METHOD getNewBBSTree :CNM_ReturnTypes.SingleExecutionResult
VAR_INPUT
	(*optional custom comparator*)
	comparator : CNM_AbstractObject.IComparator := 0;
END_VAR
VAR_OUTPUT
	(* the created tree *)
	tree :CNM_CollectionInterfaces.IBalancedBinarySearchTree;
END_VAR 
VAR
	newBalancedBinarySearchTree 	:POINTER TO BalancedBinarySearchTree;
END_VAR
VAR CONSTANT
	OBJECT_NOT_REFERENCED 			:__XWORD		:= 0;
END_VAR
getNewBBSTree := CNM_ReturnTypes.SingleExecutionResult.ERROR;
IF THIS^.isObjectValid(comparator) THEN
	newBalancedBinarySearchTree := __NEW(
	BalancedBinarySearchTree(nodeComparator := comparator)
	);
ELSE
	newBalancedBinarySearchTree := __NEW(
	BalancedBinarySearchTree(nodeComparator := OBJECT_NOT_REFERENCED)
	);
END_IF

IF (newBalancedBinarySearchTree <> 0) THEN
	tree := newBalancedBinarySearchTree^;
	getNewBBSTree := CNM_ReturnTypes.SingleExecutionResult.SUCCESS;
END_IF
END_METHOD

(*

## Short summary

function to create a new balanced binary searchtree node

.. <legal notes>

legal notes
=================
| SPDX-FileCopyrightText: © 2022 ekvip automation GmbH <info@ekvip.de>
| SPDX-License-Identifier: Apache-2.0
| For details check: Apache-2.0_

.. _Apache-2.0: https://www.apache.org/licenses/LICENSE-2.0

.. </legal notes>


**Return:** ``SingleExecutionResult.SUCCESS``: allocation succesful, output node contains new tree node instance
    ``SingleExecutionResult.ERROR``: error during allocation, output node is NULL

*)

METHOD getNewBBSTreeNode :CNM_ReturnTypes.SingleExecutionResult 
VAR_INPUT
	(* the object that should be wrapped *)
	object :CNM_AbstractObject.IObject;
END_VAR
VAR_OUTPUT
	(* the created tree node container element *)
	node :CNM_CollectionInterfaces.IBalancedBinarySearchTreeNode;
END_VAR
VAR 
	newTreeNode 		:POINTER TO BalancedBinarySearchTreeNode;
END_VAR
VAR CONSTANT
	IS_NOT_REFERENCED 	:__XWORD := 0;
END_VAR
getNewBBSTreeNode := CNM_ReturnTypes.SingleExecutionResult.ERROR;
newTreeNode := __NEW(
	BalancedBinarySearchTreeNode(
		value := object,
		left := IS_NOT_REFERENCED,
		right := IS_NOT_REFERENCED
	)
);
IF (newTreeNode <> 0) THEN
	newTreeNode^.leftChild := IS_NOT_REFERENCED;
	newTreeNode^.rightChild := IS_NOT_REFERENCED;
	node := newTreeNode^;
	getNewBBSTreeNode := CNM_ReturnTypes.SingleExecutionResult.SUCCESS;
END_IF
END_METHOD

(*

## Short summary

Method to create new Instance of DoublyLinkedElements and automatically link with other ellements.
This will affect/change the next and previouse elements !

.. <legal notes>

legal notes
=================
| SPDX-FileCopyrightText: © 2022 ekvip automation GmbH <info@ekvip.de>
| SPDX-License-Identifier: Apache-2.0
| For details check: Apache-2.0_

.. _Apache-2.0: https://www.apache.org/licenses/LICENSE-2.0

.. </legal notes>


**Return:** ``SingleExecutionResult.SUCCESS``: allocation succesful, output element contains new list element instance
    ``SingleExecutionResult.ERROR``: error during allocation, output element is NULL

*)

METHOD getNewDoublyLinkedElement :CNM_ReturnTypes.SingleExecutionResult
VAR_INPUT
	(*the dataobject to be contained inside the element*)
	object					:CNM_AbstractObject.IObject;
	(*the previous element to link to*)
	previousElement			:CNM_CollectionInterfaces.IDoublyLinkedElement;
	(*the next element to link to*)
	nextElement				:CNM_CollectionInterfaces.IDoublyLinkedElement;	
	(*a flag if the link to next and previous should be created*)
	linkElements			:BOOL := TRUE;
END_VAR
VAR_OUTPUT
	(* the created array linked list container element *)
	element :CNM_CollectionInterfaces.IDoublyLinkedElement;
END_VAR
VAR
	newElement		:POINTER TO DoublyLinkedElement;
END_VAR
getNewDoublyLinkedElement := CNM_ReturnTypes.SingleExecutionResult.ERROR;
newElement := __NEW(
	DoublyLinkedElement(
		content		:= object,
		previous	:= previousElement,
		next		:= nextElement
	)
);

IF (newElement <> 0) THEN
	IF (linkElements) THEN
		IF (THIS^.isObjectValid(previousElement)) THEN
			previousElement.next := newElement^;
		END_IF
		IF (THIS^.isObjectValid(nextElement)) THEN
			nextElement.previous := newElement^;
		END_IF	
	END_IF
	element := newElement^;
	getNewDoublyLinkedElement := CNM_ReturnTypes.SingleExecutionResult.SUCCESS;
END_IF
END_METHOD

(*

## Short summary

A method to generate a new LinkedList.

.. <legal notes>

legal notes
=================
| SPDX-FileCopyrightText: © 2022 ekvip automation GmbH <info@ekvip.de>
| SPDX-License-Identifier: Apache-2.0
| For details check: Apache-2.0_

.. _Apache-2.0: https://www.apache.org/licenses/LICENSE-2.0

.. </legal notes>



*)

METHOD getNewLinkedList :CNM_ReturnTypes.SingleExecutionResult
VAR_OUTPUT
	(* the created linked list *)
	list :CNM_CollectionInterfaces.ILinkedList;
END_VAR
VAR
	newList	:POINTER TO LinkedList;
END_VAR
getNewLinkedList := CNM_ReturnTypes.SingleExecutionResult.ERROR;
newList := __NEW(
	LinkedList()
);
IF (newList <> 0) THEN
	list := newList^;
	getNewLinkedList := CNM_ReturnTypes.SingleExecutionResult.SUCCESS;
END_IF
END_METHOD

(*

## Short summary

This method will create a new MergeSorter for linked lists.

.. <legal notes>

legal notes
=================
| SPDX-FileCopyrightText: © 2025 ekvip automation GmbH <info@ekvip.de>
| SPDX-License-Identifier: Apache-2.0
| For details check: Apache-2.0_

.. _Apache-2.0: https://www.apache.org/licenses/LICENSE-2.0

.. </legal notes>



*)
METHOD getNewLinkedListMergeSorter : CNM_CollectionInterfaces.CNM_ReturnTypes.SingleExecutionResult
VAR_OUTPUT
	(* the created linked list merge sorter *)
	sorter	: CNM_CollectionInterfaces.ILinkedListSorter;
END_VAR
VAR
	newMergeSorter :POINTER TO LinkedListMergeSorter; 
END_VAR
getNewLinkedListMergeSorter := CNM_ReturnTypes.SingleExecutionResult.ERROR;
newMergeSorter := __NEW(LinkedListMergeSorter());

IF (newMergeSorter <> 0) THEN
	sorter := newMergeSorter^;
	getNewLinkedListMergeSorter := CNM_ReturnTypes.SingleExecutionResult.SUCCESS;
END_IF
END_METHOD

END_FUNCTION_BLOCK

// ---- Lists/ArrayList/ArrayListSorter/ArrayListMergeSorter.TcPOU
(*

## Short summary

This FB sorts the list using a mergesort, which has O(n*log(n)) runtime. 
For random data it is a bit faster than Timsort, else Timsort should be used. Needs to allocate extra memory while sorting, same size as currentContainerSize.

**Caution:**
	Due to the characteristics of a merge, a merge must be performed atomically.
	As a merge of two lists l1 and l2 can take up to l1.size compares.
	That implies that at the last cycle of the merge, an atomic operation that requires up to list.size/2 compares must be performed.
	Therefore the maxCycleCompares may be exceeded and set the maxCycleCompares to a value smaller than list.size/2 may not have the desired effect.
	
.. <legal notes>

legal notes
=================
| SPDX-FileCopyrightText: © 2022 ekvip automation GmbH <info@ekvip.de>
| SPDX-License-Identifier: Apache-2.0
| For details check: Apache-2.0_

.. _Apache-2.0: https://www.apache.org/licenses/LICENSE-2.0

.. </legal notes>



*)

{attribute 'enable_dynamic_creation'}
FUNCTION_BLOCK FINAL ArrayListMergeSorter EXTENDS AbstractMergeBasedSorter
VAR
	sortBuffer :POINTER TO CNM_AbstractObject.IObject;
END_VAR


(*

## Short summary

This abstract property returns the class name of the concrete object, 
which is useful to check the class name for ``__DELETE``.

.. <legal notes>

legal notes
=================
| SPDX-FileCopyrightText: © 2022 ekvip automation GmbH <info@ekvip.de>
| SPDX-License-Identifier: Apache-2.0
| For details check: Apache-2.0_

.. _Apache-2.0: https://www.apache.org/licenses/LICENSE-2.0

.. </legal notes>

*)
PROPERTY className	:CNM_AbstractObject.ClassName
GET
className := 'CNM_Collections.ArrayListMergeSorter';
END_GET
END_PROPERTY


(*

## Short summary

This method is used to create a new instance
of the object which has the same internal state as the object.
If the object is a container class, the references to the content objects
are not cloned for this there is the method ``ICloneable.deepClone``.

If an object does not support cloning the return value is
``CNM_ReturnTypes.CloneResult.CLONE_IS_NOT_SUPPORTED``.

If there is not enough memory or the cloning fails because the
attribute enable dynamic creation was forgotten the return value is 
``CNM_ReturnTypes.CloneResult.FAILED``.

Only if the return value is ``CNM_ReturnTypes.CloneResult.SUCCESS``
the output ``clonedObject`` points to the new object
otherwise ``clonedObject`` is NULL.  

.. <legal notes>

legal notes
=================
| SPDX-FileCopyrightText: © 2022 ekvip automation GmbH <info@ekvip.de>
| SPDX-License-Identifier: Apache-2.0
| For details check: Apache-2.0_

.. _Apache-2.0: https://www.apache.org/licenses/LICENSE-2.0

.. </legal notes>


**Return:**	``CNM_ReturnTypes.CloneResult.SUCCESS``: new object clone was created,
	``CNM_ReturnTypes.CloneResult.FAILED``: object clone failed
	``CNM_ReturnTypes.CloneResult.CLONE_IS_NOT_SUPPORTED``: object does not support cloning

*)
METHOD clone	:CNM_AbstractObject.CNM_ReturnTypes.CloneResult
VAR_OUTPUT
	(* new object instance or NULL if somthing went wrong *)
	clonedObject	:CNM_AbstractObject.IObject;
END_VAR
VAR
	newSorter :POINTER TO ArrayListMergeSorter;
	sorter :CNM_CollectionInterfaces.IArrayListSorter;
END_VAR
newSorter := __NEW(
	ArrayListMergeSorter()
);

IF (newSorter = 0) THEN
	clone := CNM_ReturnTypes.CloneResult.FAILED;
ELSE
	clone := CNM_ReturnTypes.CloneResult.SUCCESS;
	THIS^.prepareClonedSorter(newSorter^);
	clonedObject := newSorter^;
END_IF
END_METHOD

(*

## Short summary

Mark the object as deleted, as it staiys in the memory.

.. <legal notes>

legal notes
=================
| SPDX-FileCopyrightText: © 2022 ekvip automation GmbH <info@ekvip.de>
| SPDX-License-Identifier: Apache-2.0
| For details check: Apache-2.0_

.. _Apache-2.0: https://www.apache.org/licenses/LICENSE-2.0

.. </legal notes>

*)
METHOD FB_Exit : BOOL
VAR_INPUT
	(* TRUE: the exit method is called in order to leave the instance which will be copied afterwards (online change).*)
	bInCopyCode	: BOOL;
END_VAR
IF THIS^.sortBuffer <> 0  THEN
	__DELETE(THIS^.sortBuffer);	
END_IF
END_METHOD

(*

## Short summary

This method sorts the data structure instantly within one call. 
It uses the passed Comparator to sort the structure or the compareTo of the contained Objects if no comparator is passed.

.. <legal notes>

legal notes
=================
| SPDX-FileCopyrightText: © 2022 ekvip automation GmbH <info@ekvip.de>
| SPDX-License-Identifier: Apache-2.0
| For details check: Apache-2.0_

.. _Apache-2.0: https://www.apache.org/licenses/LICENSE-2.0

.. </legal notes>


**Return:**``ERROR``: Sort was not able to finish 
	``SUCCESS``: Sorting was finished succesfully

*)
METHOD instantSort : CNM_CollectionInterfaces.CNM_ReturnTypes.SingleExecutionResult
VAR_INPUT
	(*The size of the list to be sorted*)
	size	: UDINT;
	(*the container, that contains the list elements*)
	container	: POINTER TO CNM_CollectionInterfaces.CNM_AbstractObject.IObject;
	(*the comparator that should be used for the sort. Must not be changed while sort is in process*)
	comparator	: CNM_CollectionInterfaces.CNM_AbstractObject.IComparator := 0;
END_VAR
VAR_IN_OUT
	(*the current version of the list, must change when the data in the list changes *)
	currentListVersion	: __XWORD;
END_VAR
VAR 
	instantSortBuffer :POINTER TO CNM_AbstractObject.IObject;
	currentSortSize 	:UDINT := 1;
	leftBound 			:UDINT;
	middle 				:UDINT;
	rightBound 			:UDINT;
	maximumLeftBound	:UDINT;
	stepSize 			:UDINT;
END_VAR
VAR CONSTANT
	NULL :__XWORD := 0;
END_VAR
instantSortBuffer := __NEW(__XWORD, size);
THIS^.setComparator(comparator);
WHILE (currentSortSize <= size-1) DO
	maximumLeftBound := size -2;
	stepSize := 2*currentSortSize;
	FOR leftBound := 0 TO maximumLeftBound BY (stepSize) DO
		
		IF leftBound+currentSortSize-1 < size-1 THEN
			middle := leftBound + currentSortSize-1;
		ELSE
			middle := size-1;
		END_IF
		IF leftBound + stepSize - 1 < size THEN
			rightBound := leftBound + stepSize -1;
		ELSE
			rightBound := size-1;
		END_IF
		
		instantSort := merge(
			firstContainer := ADR(container[leftBound]),
			secondContainer := ADR(container[middle + 1]),
			buffer := instantSortBuffer,
			firstContainerSize := middle - leftBound + 1,
			secondContainerSize := rightBound - middle 
		);
		IF instantSort <> CNM_ReturnTypes.SingleExecutionResult.SUCCESS THEN
			__DELETE(instantSortBuffer);
			RETURN;
		END_IF
		
		Tc2_System.MEMMOVE(
			destAddr := ADR(container[leftBound]),
			srcAddr := THIS^.sortBuffer,
			n := rightBound - leftBound + 1
		);
	END_FOR
END_WHILE

currentListVersion := currentListVersion + 1;
instantSort := CNM_ReturnTypes.SingleExecutionResult.SUCCESS;
END_METHOD

(*

## Short summary

This method sorts the data structure. 
It uses the passed Comperator to sort the structure.
This can take many cycles and should be called until the CNM_ReturnTypes.ExecutionState is no longer ``BUSY``.

.. <legal notes>

legal notes
=================
| SPDX-FileCopyrightText: © 2022 ekvip automation GmbH <info@ekvip.de>
| SPDX-License-Identifier: Apache-2.0
| For details check: Apache-2.0_

.. _Apache-2.0: https://www.apache.org/licenses/LICENSE-2.0

.. </legal notes>


**Return:** ``ABORTED``: While sort was pending,execute had a falling edge,
	``BUSY``: Sort is in progress
	``ERROR``: Sort was not able to finish (p.e. List changed) call sort(false) to reset
	``IDLE``: Currently no sort in progress
	``SUCCESS``: Sorting was finished 

*)
METHOD sort	:CNM_ReturnTypes.SingleExecutionState
VAR_INPUT
	(*control bit to start or abort the sorting, needs to be active until the ExecutionState is SUCCESS*)
	execute		:BOOL;
	(*The size of the list to be sorted*)
	size 		:UDINT;
	(*the container, that contains the list elements*)
	container	:POINTER TO CNM_AbstractObject.IObject;
	(*the comparator that should be used for the sort. Must not be changed while sort is in process*)
	comparator	:CNM_AbstractObject.IComparator		:= 0;
END_VAR
VAR_IN_OUT
	(*the current version of the list, must change when the data in the list changes *)
	currentListVersion :__XWORD;
END_VAR
VAR_INST
	cycleManager :CNM_CycleManager.SimpleCycleManager;
	lastExecute			:BOOL		:= FALSE;
	executing 			:BOOL		:= FALSE;
	state 				:CNM_ReturnTypes.SingleExecutionState	:= CNM_ReturnTypes.SingleExecutionState.IDLE; 
	currentSortSize 	:UDINT;
	startAt 			:UDINT 	:= 0;
	(* list version index, used to detect list changes during sorting *)
	lastListChangeIndex :__XWORD;
END_VAR
VAR 
	leftBound 			:UDINT;
	middle 				:UDINT;
	rightBound 			:UDINT;
	operationsThisCycle	:UDINT :=0;
	leave 				:BOOL := FALSE;
	mergeState 			:CNM_ReturnTypes.SingleExecutionResult;
	maximumLeftBound	:UDINT;
	stepSize 			:UDINT;
END_VAR
VAR CONSTANT
	INIT :DINT := CNM_ReturnTypes.DefaultSteps.STEP.INIT;
	SORT_LIST :DINT := INIT + 1;
	CLEAN_UP :DINT := SORT_LIST + 1;
	ERROR :DINT := CNM_ReturnTypes.DefaultSteps.STEP.ERROR;
	REGISTER_SIZE :UDINT := SIZEOF(__XWORD);
END_VAR
cycleManager(execute := execute);
IF cycleManager.step.current > INIT THEN
	cycleManager.assert.bitNumber.x.valueIsEqualTo(
		currentValue := currentListVersion, 
		expectedValue := lastListChangeIndex, 
		message := 'list has changed during pending sorting'
	);
END_IF


CASE cycleManager.step.current OF
INIT:
	cycleManager.configuration.sequence.requireSuccessStep := FALSE;
	THIS^.setComparator(comparator);
	lastListChangeIndex := currentListVersion;
	startAt := 0;
	IF size > 1 THEN
		currentSortSize := 1;
		__DELETE(THIS^.sortBuffer);
		THIS^.sortBuffer := __NEW(__XWORD, size);
		THIS^.maxOperationsPerCycle := size;
		cycleManager.proceed();
	ELSE
		cycleManager.proceedWith(step := CNM_ReturnTypes.DefaultSteps.STEP.SUCCESS);
	END_IF
	
SORT_LIST:
	IF (lastListChangeIndex <> currentListVersion) THEN
		cycleManager.proceedWith(ERROR);
		sort := CNM_ReturnTypes.SingleExecutionState.ERROR;
		RETURN;
	END_IF
	IF currentSortSize <= size-1 THEN
		WHILE (operationsThisCycle < THIS^.maxCycleCompares) DO
			maximumLeftBound := size -2;
			stepSize := 2*currentSortSize;
			FOR leftBound := startAt TO maximumLeftBound BY (stepSize) DO
				IF (operationsThisCycle > THIS^.maxCycleCompares) THEN
					leave := TRUE;
					EXIT;
				END_IF
				
				IF leftBound+currentSortSize-1 < size-1 THEN
					middle := leftBound + currentSortSize-1;
				ELSE
					middle := size-1;
				END_IF
				IF leftBound + stepSize - 1 < size THEN
					rightBound := leftBound + stepSize -1;
				ELSE
					rightBound := size-1;
				END_IF
				
				mergeState := merge(
					firstContainer := ADR(container[leftBound]),
					secondContainer := ADR(container[middle + 1]),
					buffer := THIS^.sortBuffer,
					firstContainerSize := middle - leftBound + 1,
					secondContainerSize := rightBound - middle 
				);
				IF mergeState <> CNM_ReturnTypes.SingleExecutionResult.SUCCESS THEN
					cycleManager.proceedWith(CNM_ReturnTypes.DefaultSteps.STEP.ERROR);
					sort := CNM_ReturnTypes.SingleExecutionState.ERROR;
					RETURN;
				END_IF
				Tc2_System.MEMMOVE(
					destAddr := ADR(container[leftBound]),
					srcAddr := THIS^.sortBuffer,
					n := (rightBound - leftBound + 1) * REGISTER_SIZE
				);
				operationsThisCycle := operationsThisCycle + stepSize - 1;
				
			END_FOR
			
			IF leave THEN
				startAt := leftBound;
				EXIT;
			ELSE
				startAt := 0;
				currentSortSize := stepSize;
				IF currentSortSize > size-1 THEN
					EXIT;
				END_IF
			END_IF
		END_WHILE
	END_IF

	//check if sort done within same cycle
	IF currentSortSize > size-1 THEN 
		cycleManager.proceedWith(CNM_ReturnTypes.DefaultSteps.STEP.SUCCESS);
		IF THIS^.sortBuffer <> 0  THEN
			__DELETE(sortBuffer);	
		END_IF
	END_IF
	
	lastListChangeIndex := currentListVersion := currentListVersion + 1;
	
CLEAN_UP,
CNM_ReturnTypes.DefaultSteps.STEP.ERROR,
CNM_ReturnTypes.DefaultSteps.STEP.ABORT,
CNM_ReturnTypes.DefaultSteps.STEP.SUCCESS:
	IF THIS^.sortBuffer <> 0  THEN
		__DELETE(sortBuffer);	
	END_IF
	
END_CASE
sort := cycleManager.state;
END_METHOD

END_FUNCTION_BLOCK

// ---- Lists/ArrayList/ArrayListSorter/AbstractMergeBasedSorter.TcPOU
(*

## Short summary

Abstract Sorter for merge based sort methods. 
Provides a default implementation for an indexed merge function and a method to efficient copy elements.

**Caution:**
	Due to the characteristics of a merge, a merge must be performed atomically.
	As a merge of two lists l1 and l2 can take up to l1.size+l2.size-1 compares.
	That implies that at the last cycle of the merge, an atomic operation that requires up to list.size-1 compares must be performed.
	Therefore the maxCycleCompares may be exceeded and set the maxCycleCompares to a value smaller than list.size-1 may not have the desired effect.
 
.. <legal notes>

legal notes
=================
| SPDX-FileCopyrightText: © 2022 ekvip automation GmbH <info@ekvip.de>
| SPDX-License-Identifier: Apache-2.0
| For details check: Apache-2.0_

.. _Apache-2.0: https://www.apache.org/licenses/LICENSE-2.0

.. </legal notes>



*)

FUNCTION_BLOCK INTERNAL ABSTRACT AbstractMergeBasedSorter EXTENDS AbstractArrayListSorter

(*

## Short summary

Function that sorts specified parts using a merge mechanism.
Writes the result into a given buffer. 
Buffer size must be at least as big as both given containers combined.

.. <legal notes>

legal notes
=================
| SPDX-FileCopyrightText: © 2025 ekvip automation GmbH <info@ekvip.de>
| SPDX-License-Identifier: Apache-2.0
| For details check: Apache-2.0_

.. _Apache-2.0: https://www.apache.org/licenses/LICENSE-2.0

.. </legal notes>


**Return:** CNM_ReturnTypes.ExecutionResult: the result of the merge,
	ERROR if any parameter was invalid for merge 
	SUCCESS if list is merged and result in buffer

*)

METHOD PROTECTED FINAL merge : CNM_ReturnTypes.SingleExecutionResult
VAR_INPUT
	firstContainer :POINTER TO CNM_AbstractObject.IObject;
	secondContainer :POINTER TO CNM_AbstractObject.IObject;
	buffer :POINTER TO CNM_AbstractObject.IObject;
	firstContainerSize :UDINT;
	secondContainerSize :UDINT;
END_VAR
VAR
	leftIndex :UDINT;
	rightIndex :UDINT;
	destination :__XWORD;
	source :__XWORD;
	remainingElements :UDINT;
END_VAR
VAR CONSTANT
	REGISTER_SIZE :UDINT := SIZEOF(__XWORD);
END_VAR
merge := CNM_ReturnTypes.SingleExecutionResult.ERROR;
RETURN (
	(buffer = 0)
	OR_ELSE (firstContainer = 0) 
	OR_ELSE (secondContainer = 0)
	OR_ELSE (firstContainer = secondContainer)
);

merge := CNM_ReturnTypes.SingleExecutionResult.SUCCESS;
RETURN (
	((firstContainerSize + secondContainerSize) = 0) 
);

WHILE(
	(rightIndex < secondContainerSize) 
	AND_THEN (leftIndex < firstContainerSize)
)DO
	IF ( 
		THIS^.compareElements(
			firstContainer[leftIndex],secondContainer[rightIndex]
		) <= CNM_ReturnTypes.ComparationResult.EQUAL
	) THEN
		buffer[leftIndex+rightIndex] := firstContainer[leftIndex];
		leftIndex := leftIndex + 1;
	ELSE
		buffer[leftIndex+rightIndex] := secondContainer[rightIndex];
		rightIndex := rightIndex + 1;
	END_IF
END_WHILE

destination := ADR(buffer[leftIndex+rightIndex]);
IF(leftIndex = firstContainerSize)THEN
	source := ADR(secondContainer[rightIndex]);
	remainingElements := secondContainerSize - rightIndex;
ELSE
	source := ADR(firstContainer[leftIndex]);
	remainingElements := firstContainerSize - leftIndex;
END_IF

Tc2_System.MEMMOVE(
	destAddr := destination,
	srcAddr := source,
	n := remainingElements * REGISTER_SIZE
);
END_METHOD

END_FUNCTION_BLOCK

// ---- Lists/Sorter/classes/AbstractArrayListSorter.TcPOU
(*

## Short summary

The abstract implementation of an ArrayListSorter, to provide default implementations for setting comparator, the IObject methods.
Provides the default implementation for sort and inverseSort.

.. <legal notes>

legal notes
=================
| SPDX-FileCopyrightText: © 2022 ekvip automation GmbH <info@ekvip.de>
| SPDX-License-Identifier: Apache-2.0
| For details check: Apache-2.0_

.. _Apache-2.0: https://www.apache.org/licenses/LICENSE-2.0

.. </legal notes>



*)

FUNCTION_BLOCK INTERNAL ABSTRACT AbstractArrayListSorter EXTENDS AbstractListSorter IMPLEMENTS CNM_CollectionInterfaces.IArrayListSorter

(*

## Short summary

This method sorts the data structure instantly in descending order within one call. 
It uses the passed Comparator to sort the structure or the compareTo of the contained Objects if no comparator is passed.

.. <legal notes>

legal notes
=================
| SPDX-FileCopyrightText: © 2022 ekvip automation GmbH <info@ekvip.de>
| SPDX-License-Identifier: Apache-2.0
| For details check: Apache-2.0_

.. _Apache-2.0: https://www.apache.org/licenses/LICENSE-2.0

.. </legal notes>


**Return:**``ERROR``: Sort was not able to finish 
	``SUCCESS``: Sorting was finished succesfully

*)
METHOD instantInverseSort : CNM_CollectionInterfaces.CNM_ReturnTypes.SingleExecutionResult
VAR_INPUT
	(*The size of the list to be sorted*)
	size	: UDINT;
	(*the container, that contains the list elements*)
	container	: POINTER TO CNM_CollectionInterfaces.CNM_AbstractObject.IObject;
	(*the comparator that should be used for the sort. Must not be changed while sort is in process*)
	comparator	: CNM_CollectionInterfaces.CNM_AbstractObject.IComparator := 0;
END_VAR
VAR_IN_OUT
	(*the current version of the list, must change when the data in the list changes *)
	currentListVersion	: __XWORD;
END_VAR
THIS^.reverseComparator.attachComparator(comparator);
THIS^.instantSort(size := size, comparator := THIS^.reverseComparator, container := container, currentListVersion := currentListVersion);
END_METHOD

(*

## Short summary

This method sorts the data structure instantly within one call. 
It uses the passed Comparator to sort the structure or the compareTo of the contained Objects if no comparator is passed.

.. <legal notes>

legal notes
=================
| SPDX-FileCopyrightText: © 2022 ekvip automation GmbH <info@ekvip.de>
| SPDX-License-Identifier: Apache-2.0
| For details check: Apache-2.0_

.. _Apache-2.0: https://www.apache.org/licenses/LICENSE-2.0

.. </legal notes>


**Return:**``ERROR``: Sort was not able to finish 
	``SUCCESS``: Sorting was finished succesfully

*)
METHOD ABSTRACT instantSort : CNM_CollectionInterfaces.CNM_ReturnTypes.SingleExecutionResult
VAR_INPUT
	(*The size of the list to be sorted*)
	size	: UDINT;
	(*the container, that contains the list elements*)
	container	: POINTER TO CNM_CollectionInterfaces.CNM_AbstractObject.IObject;
	(*the comparator that should be used for the sort. Must not be changed while sort is in process*)
	comparator	: CNM_CollectionInterfaces.CNM_AbstractObject.IComparator := 0;
END_VAR
VAR_IN_OUT
	(*the current version of the list, must change when the data in the list changes *)
	currentListVersion	: __XWORD;
END_VAR
END_METHOD


(*

## Short summary

This method sorts the Sortable in the inverted order, so from great to low
.. <legal notes>

legal notes
=================
| SPDX-FileCopyrightText: © 2025 ekvip automation GmbH <info@ekvip.de>
| SPDX-License-Identifier: Apache-2.0
| For details check: Apache-2.0_

.. _Apache-2.0: https://www.apache.org/licenses/LICENSE-2.0

.. </legal notes>


**Return:** ``ABORTED``: While inverse was pending,execute had a falling edge,
	``BUSY``: Inverse is in progress
	``ERROR``: Inverse was not able to finish (p.e. List changed) call inverse(false) to reset
	``IDLE``: Currently invert is not in progress
	``SUCCESS``: Inversing was finished 
*)
METHOD inverseSort : CNM_ReturnTypes.SingleExecutionState
VAR_INPUT
	(*control bit to start or abort the inverting, needs to be active until the ExecutionState is noz longer busy*)
	execute	: BOOL;
	(*The size of the list to be sorted*)
	size :UDINT;
	(*the container, that contains the list elements*)
	container	: POINTER TO CNM_AbstractObject.IObject;
END_VAR
VAR_INPUT
	(*the comparator that should be used for the sort. Must not be changed while sort is in process*)
	comparator :CNM_AbstractObject.IComparator := 0;
END_VAR
VAR_IN_OUT
	(*the current version of the list, must change when the data in the list changes *)
	currentListVersion :__XWORD;
END_VAR
THIS^.reverseComparator.attachComparator(comparator);
THIS^.sort(execute := execute, size := size, comparator := THIS^.reverseComparator, container := container, currentListVersion := currentListVersion);
END_METHOD

(*

## Short summary

This method sorts the data structure. 
This can take many cycles and should be called until the CNM_ReturnTypes.ExecutionState is no longer ``BUSY``.

.. <legal notes>

legal notes
=================
| SPDX-FileCopyrightText: © 2025 ekvip automation GmbH <info@ekvip.de>
| SPDX-License-Identifier: Apache-2.0
| For details check: Apache-2.0_

.. _Apache-2.0: https://www.apache.org/licenses/LICENSE-2.0

.. </legal notes>


**Return:** ``ABORTED``: While sort was pending,execute had a falling edge,
	``BUSY``: Sort is in progress
	``ERROR``: Sort was not able to finish (p.e. List changed) call sort(false) to reset
	``IDLE``: Currently no sort in progress
	``SUCCESS``: Sorting was finished 

*)
METHOD ABSTRACT sort :CNM_ReturnTypes.SingleExecutionState
VAR_INPUT
	(*control bit to start or abort the sorting, needs to be active until the ExecutionState is SUCCESS*)
	execute		:BOOL;
	(*The size of the list to be sorted*)
	size 		:UDINT;
	(*the container, that contains the list elements*)
	container	:POINTER TO CNM_AbstractObject.IObject;
	(*the comparator that should be used for the sort. Must not be changed while sort is in process*)
	comparator :CNM_AbstractObject.IComparator := 0;
END_VAR
VAR_IN_OUT
	(*the current version of the list, must change when the data in the list changes *)
	currentListVersion :__XWORD;
END_VAR
END_METHOD

END_FUNCTION_BLOCK

// ---- Lists/Sorter/classes/AbstractListSorter.TcPOU
(*

## Short summary

Abstract base class for list sorters. Provides functionality to set the execution limits, size and list changes.

.. <legal notes>

legal notes
=================
| SPDX-FileCopyrightText: © 2023 ekvip automation GmbH <info@ekvip.de>
| SPDX-License-Identifier: Apache-2.0
| For details check: Apache-2.0_

.. _Apache-2.0: https://www.apache.org/licenses/LICENSE-2.0

.. </legal notes>



*)

FUNCTION_BLOCK INTERNAL ABSTRACT AbstractListSorter EXTENDS AbstractDisposableContainer IMPLEMENTS CNM_CollectionInterfaces.IListSorter
VAR
	(*The comparator used to sort, set by the List when setting sorter*)
	elementComparator		:CNM_AbstractObject.IComparator;
	(*The maximum of comparisons that the sorter allows, may be overwruled by the bounds*)
	maxOperationsPerCycle 	:UDINT;
	(*The maximum of compares done per cycle to prevent very long lists to take up to much time*)
	upperCompareBound 		:UDINT	:= GeneralParameters.DEFAULT_OPERATIONS_PER_CYCLE;
	(* Comparator used for inverse Sort *)
	reverseComparator :InvertComparator;
	(* the current change index of the list *)
	listChangeIndex :REFERENCE TO __XWORD;
END_VAR


(*

## Short summary

This abstract property returns the class name of the concrete object, 
which is useful to check the class name for ``__DELETE``.

.. <legal notes>

legal notes
=================
| SPDX-FileCopyrightText: © 2022 ekvip automation GmbH <info@ekvip.de>
| SPDX-License-Identifier: Apache-2.0
| For details check: Apache-2.0_

.. _Apache-2.0: https://www.apache.org/licenses/LICENSE-2.0

.. </legal notes>

*)
PROPERTY ABSTRACT className	:CNM_AbstractObject.ClassName
GET
END_GET
END_PROPERTY

(*

## Short summary

This method is called in the destruct method and is intended to zero all references and interfaces that should not be destructed. 
To delete the collection with all its contents, use deepDestruct() instead of destruct().

.. <legal notes>

legal notes
=================
| SPDX-FileCopyrightText: © 2025 ekvip automation GmbH <info@ekvip.de>
| SPDX-License-Identifier: Apache-2.0
| For details check: Apache-2.0_

.. _Apache-2.0: https://www.apache.org/licenses/LICENSE-2.0

.. </legal notes>

*)
METHOD PROTECTED clearContents
THIS^.elementComparator := 0;
END_METHOD


(*

## Short summary

This method is used to create a new instance
of the object which has the same internal state as the object.
If the object is a container class, the references to the content objects
are not cloned for this there is the method `ICloneable.deepClone`.

If an object does not support cloning the return value is
``CNM_ReturnTypes.CloneResult.CLONE_IS_NOT_SUPPORTED``.

If there is not enough memory or the cloning fails because the
attribute enable dynamic creation was forgotten the return value is 
``CNM_ReturnTypes.CloneResult.FAILED``.

Only if the return value is ``CNM_ReturnTypes.CloneResult.SUCCESS``
the output ``clonedObject`` points to the new object
otherwise ``clonedObject`` is NULL.  

.. <legal notes>

legal notes
=================
| SPDX-FileCopyrightText: © 2022 ekvip automation GmbH <info@ekvip.de>
| SPDX-License-Identifier: Apache-2.0
| For details check: Apache-2.0_

.. _Apache-2.0: https://www.apache.org/licenses/LICENSE-2.0

.. </legal notes>


**Return:** ``CNM_ReturnTypes.CloneResult.SUCCESS``: new object clone was created,
    ``CNM_ReturnTypes.CloneResult.FAILED``: object clone failed
    ``CNM_ReturnTypes.CloneResult.CLONE_IS_NOT_SUPPORTED``: object does not support cloning

*)

METHOD ABSTRACT clone	:CNM_AbstractObject.CNM_ReturnTypes.CloneResult
VAR_OUTPUT
	(* new object instance or NULL if somthing went wrong *)
	clonedObject	:CNM_AbstractObject.IObject;
END_VAR
END_METHOD

(*

## Short summary

Compares two objects, if set uses the comparator, else uses the built in comparator of object1.

.. <legal notes>

legal notes
=================
| SPDX-FileCopyrightText: © 2022 ekvip automation GmbH <info@ekvip.de>
| SPDX-License-Identifier: Apache-2.0
| For details check: Apache-2.0_

.. _Apache-2.0: https://www.apache.org/licenses/LICENSE-2.0

.. </legal notes>


**Return:** ``Smaller``: ``Object1`` precendes ``Object2`` in order,
	``Greater``: ``Object1`` succeds ``Object2`` in order,
	``Equal``: ``Object1`` equals ``Object2`` in Order
	
*)

METHOD PROTECTED compareElements	:CNM_ReturnTypes.ComparationResult
VAR_INPUT
	(*first object to compare*)
	object1	:CNM_AbstractObject.IObject;
	(*second object to compare*)
	object2	:CNM_AbstractObject.IObject;
END_VAR
IF THIS^.isObjectValid(THIS^.elementComparator) THEN 
	compareElements := THIS^.elementComparator.compare(object1,object2);   
ELSIF (THIS^.isObjectValid(object1)) THEN
	compareElements := object1.compareTo(object2);
ELSIF (THIS^.isObjectValid(object2)) THEN
	compareElements := CNM_ReturnTypes.ComparationResult.GREATER;
ELSE
	compareElements := CNM_ReturnTypes.ComparationResult.EQUAL;
END_IF
END_METHOD


(*

## Short summary

This method is used to create a new instance
of the object which has the same internal state as the object.
If the object is a container class, the references to the content objects
are cloned too.

If an object does not support cloning the return value is
``CNM_ReturnTypes.CloneResult.CLONE_IS_NOT_SUPPORTED``.

If there is not enough memory or the cloning fails because the
attribute enable dynamic creation was forgotten the return value is 
``CNM_ReturnTypes.CloneResult.FAILED``.
If something goes wrong, then this method must clean up everything
that has been cloned and free the memory again.
**The deepClone either works completely, or not at all**

Only if the return value is ``CNM_ReturnTypes.CloneResult.SUCCESS``
the output ``clonedObject`` points to the new object
otherwise ``clonedObject`` is NULL.  

.. <legal notes>

legal notes
=================
| SPDX-FileCopyrightText: © 2022 ekvip automation GmbH <info@ekvip.de>
| SPDX-License-Identifier: Apache-2.0
| For details check: Apache-2.0_

.. _Apache-2.0: https://www.apache.org/licenses/LICENSE-2.0

.. </legal notes>


**Return:** ``CNM_ReturnTypes.CloneResult.SUCCESS``: new object clone was created,
    ``CNM_ReturnTypes.CloneResult.FAILED``: object clone failed
    ``CNM_ReturnTypes.CloneResult.CLONE_IS_NOT_SUPPORTED``: object does not support deep cloning

*)

METHOD deepClone	:CNM_AbstractObject.CNM_ReturnTypes.CloneResult
VAR_OUTPUT
	(* new object instance or NULL if somthing went wrong *)
	clonedObject	:CNM_AbstractObject.IObject;
END_VAR
deepClone := THIS^.clone(clonedObject => clonedObject);
END_METHOD

(*

## Short summary

Mark the object as deleted, as it staiys in the memory.

.. <legal notes>

legal notes
=================
| SPDX-FileCopyrightText: © 2022 ekvip automation GmbH <info@ekvip.de>
| SPDX-License-Identifier: Apache-2.0
| For details check: Apache-2.0_

.. _Apache-2.0: https://www.apache.org/licenses/LICENSE-2.0

.. </legal notes>

*)
METHOD FB_Exit : BOOL
VAR_INPUT
	(* TRUE: the exit method is called in order to leave the instance which will be copied afterwards (online change).*)
	bInCopyCode	: BOOL;
END_VAR
IF THIS^.isObjectValid(THIS^.elementComparator) THEN
	THIS^.elementComparator.deepDestruct();
END_IF
END_METHOD

(*

## Short summary

This property defines the maximum amount of compares that should be done per Cycle. Is optional as default should be set by class.
Passing zero resets to class specific default.

.. <legal notes>

legal notes
=================
| SPDX-FileCopyrightText: © 2022 ekvip automation GmbH <info@ekvip.de>
| SPDX-License-Identifier: Apache-2.0
| For details check: Apache-2.0_

.. _Apache-2.0: https://www.apache.org/licenses/LICENSE-2.0

.. </legal notes>

*)

PROPERTY maxCycleCompares	:UDINT
GET
maxCycleCompares := THIS^.upperCompareBound;
END_GET
SET
THIS^.upperCompareBound := SEL(
	maxCycleCompares = 0,
	maxCycleCompares,
	GeneralParameters.DEFAULT_OPERATIONS_PER_CYCLE
);
END_SET
END_PROPERTY

(*

## Short summary

Does the basic initialization for a new sorter that was cloned from THIS^

.. <legal notes>

legal notes
=================
| SPDX-FileCopyrightText: © 2022 ekvip automation GmbH <info@ekvip.de>
| SPDX-License-Identifier: Apache-2.0
| For details check: Apache-2.0_

.. _Apache-2.0: https://www.apache.org/licenses/LICENSE-2.0

.. </legal notes>



*)

METHOD PROTECTED prepareClonedSorter
VAR_INPUT
	(*The cloned sorter to init*)
	newSorter :CNM_CollectionInterfaces.IListSorter;
END_VAR
IF (THIS^.isObjectValid(newSorter)) THEN
	newSorter.maxCycleCompares := THIS^.maxCycleCompares;	
END_IF
END_METHOD

(*

## Short summary

This method can replace the default comperator for custom one.
Useful if you par example want to invert the order of the sort.

.. <legal notes>

legal notes
=================
| SPDX-FileCopyrightText: © 2022 ekvip automation GmbH <info@ekvip.de>
| SPDX-License-Identifier: Apache-2.0
| For details check: Apache-2.0_

.. _Apache-2.0: https://www.apache.org/licenses/LICENSE-2.0

.. </legal notes>


**Return:** ``THIS^`` `IListSorter`

*)

METHOD PROTECTED setComparator	:CNM_CollectionInterfaces.IListSorter
VAR_INPUT
	(*the instance of the comperator to be used for sorting*)
	comparator	:CNM_AbstractObject.IComparator;
END_VAR
THIS^.elementComparator := comparator;
setComparator := THIS^;
END_METHOD

END_FUNCTION_BLOCK

// ---- Lists/Sorter/classes/Internal/InvertComparator.TcPOU
(*

## Short summary

Internal comparator, which returns the opposite of the .compareTo method of object1.


.. <legal notes>

legal notes
=================
| SPDX-FileCopyrightText: © 2024 ekvip automation GmbH <info@ekvip.de>
| SPDX-License-Identifier: Apache-2.0
| For details check: Apache-2.0_

.. _Apache-2.0: https://www.apache.org/licenses/LICENSE-2.0

.. </legal notes>



*)

FUNCTION_BLOCK INTERNAL InvertComparator EXTENDS CNM_AbstractObject.Object IMPLEMENTS CNM_AbstractObject.IComparator
VAR
	comparator :CNM_AbstractObject.IComparator;
END_VAR

METHOD attachComparator
VAR_INPUT
	comparator :CNM_AbstractObject.IComparator;
END_VAR
THIS^.comparator := comparator;
END_METHOD


(*

## Short summary

This abstract property returns the class name of the concrete object, 
which is useful to check the class name for ``__DELETE``.

.. <legal notes>

legal notes
=================
| SPDX-FileCopyrightText: © 2022 ekvip automation GmbH <info@ekvip.de>
| SPDX-License-Identifier: Apache-2.0
| For details check: Apache-2.0_

.. _Apache-2.0: https://www.apache.org/licenses/LICENSE-2.0

.. </legal notes>

*)
PROPERTY className : CNM_AbstractObject.ClassName
GET
className := 'CNM_Collections.InvertComparator';
END_GET
END_PROPERTY


(*

## Short summary

This method compares two objects, this is needed for sort orders.

.. <legal notes>

legal notes
=================
| SPDX-FileCopyrightText: © 2022 ekvip automation GmbH <info@ekvip.de>
| SPDX-License-Identifier: Apache-2.0
| For details check: Apache-2.0_

.. _Apache-2.0: https://www.apache.org/licenses/LICENSE-2.0

.. </legal notes>


**Return:** ``SMALLER``: ``object1`` precedes in order,
    ``EQUAL``: ``object1`` and ``object2`` at the same position in order,
    ``GREATER``: ``object1`` is after in order. Checkout the library CNM_ReturnTypes.

*)

METHOD compare : CNM_AbstractObject.CNM_ReturnTypes.ComparationResult
VAR_INPUT
	(* first object to compare*)
	object1	: CNM_AbstractObject.IObject;
	(* second object to compare*)
	object2	: CNM_AbstractObject.IObject;
END_VAR
//object2.compareTo(object1) is the inversion of object1.compareTo(object2);
IF THIS^.isObjectValid(THIS^.comparator) THEN
	compare := THIS^.comparator.compare(object2,object1); 
ELSIF (THIS^.isObjectValid(object2)) THEN
	compare := object2.compareTo(object1);
ELSIF (THIS^.isObjectValid(object1)) THEN
	compare := CNM_ReturnTypes.ComparationResult.GREATER;
ELSE
	compare := CNM_ReturnTypes.ComparationResult.EQUAL;
END_IF
END_METHOD

END_FUNCTION_BLOCK

// ---- Lists/ArrayList/ArrayListSorter/ArrayListShellSorter.TcPOU
(*

## Short summary

This FB sorts the list using a shellsort, which has O(n^(4/3)) runtime. Slower than merge or timsort but doesn't need additional memory.

.. <legal notes>

legal notes
=================
| SPDX-FileCopyrightText: © 2022 ekvip automation GmbH <info@ekvip.de>
| SPDX-License-Identifier: Apache-2.0
| For details check: Apache-2.0_

.. _Apache-2.0: https://www.apache.org/licenses/LICENSE-2.0

.. </legal notes>



*)

{attribute 'enable_dynamic_creation'}
FUNCTION_BLOCK ArrayListShellSorter EXTENDS AbstractArrayListSorter
VAR CONSTANT
	MAX_COLUMNINDEX :UINT := 7;
	//ciuras proposal for columns on shellsort
	PREPARED_COLUMN_WIDTH :ARRAY[0..MAX_COLUMNINDEX] OF __XWORD := [1,4,10,23,57,132,301,701];
END_VAR


(*

## Short summary

This abstract property returns the class name of the concrete object, 
which is useful to check the class name for ``__DELETE``.

.. <legal notes>

legal notes
=================
| SPDX-FileCopyrightText: © 2022 ekvip automation GmbH <info@ekvip.de>
| SPDX-License-Identifier: Apache-2.0
| For details check: Apache-2.0_

.. _Apache-2.0: https://www.apache.org/licenses/LICENSE-2.0

.. </legal notes>

*)
PROPERTY className :CNM_AbstractObject.ClassName
GET
className := 'CNM_Collections.ArrayListShellSorter';
END_GET
END_PROPERTY

(*

## Short summary

This method is called in the destruct method and is intended to zero all references and interfaces that should not be destructed. 
To delete the collection with all its contents, use deepDestruct() instead of destruct().

.. <legal notes>

legal notes
=================
| SPDX-FileCopyrightText: © 2025 ekvip automation GmbH <info@ekvip.de>
| SPDX-License-Identifier: Apache-2.0
| For details check: Apache-2.0_

.. _Apache-2.0: https://www.apache.org/licenses/LICENSE-2.0

.. </legal notes>

*)
METHOD PROTECTED clearContents
END_METHOD


(*

## Short summary

This method is used to create a new instance
of the object which has the same internal state as the object.
If the object is a container class, the references to the content objects
are not cloned for this there is the method ``ICloneable.deepClone``.

If an object does not support cloning the return value is
``CNM_ReturnTypes.CloneResult.CLONE_IS_NOT_SUPPORTED``.

If there is not enough memory or the cloning fails because the
attribute enable dynamic creation was forgotten the return value is 
``CNM_ReturnTypes.CloneResult.FAILED``.

Only if the return value is ``CNM_ReturnTypes.CloneResult.SUCCESS``
the output ``clonedObject`` points to the new object
otherwise ``clonedObject`` is NULL.  

.. <legal notes>

legal notes
=================
| SPDX-FileCopyrightText: © 2022 ekvip automation GmbH <info@ekvip.de>
| SPDX-License-Identifier: Apache-2.0
| For details check: Apache-2.0_

.. _Apache-2.0: https://www.apache.org/licenses/LICENSE-2.0

.. </legal notes>


**Return:** ``CNM_ReturnTypes.CloneResult.SUCCESS``: new object clone was created,
	``CNM_ReturnTypes.CloneResult.FAILED``: object clone failed
	``CNM_ReturnTypes.CloneResult.CLONE_IS_NOT_SUPPORTED``: object does not support cloning

*)
METHOD clone	:CNM_AbstractObject.CNM_ReturnTypes.CloneResult
VAR_OUTPUT
	(* new object instance or NULL if somthing went wrong *)
	clonedObject	:CNM_AbstractObject.IObject;
END_VAR
VAR
	newSorter :POINTER TO ArrayListShellSorter;
	sorter :CNM_CollectionInterfaces.IArrayListSorter;
	object :CNM_AbstractObject.IObject;
	clonedComparator :CNM_AbstractObject.IComparator;
END_VAR
newSorter := __NEW(
	ArrayListShellSorter()
);

IF (newSorter = 0) THEN
	clone := CNM_ReturnTypes.CloneResult.FAILED;
ELSE
	clone := CNM_ReturnTypes.CloneResult.SUCCESS;
	THIS^.prepareClonedSorter(newSorter^);
	clonedObject := newSorter^;
END_IF
END_METHOD

(*

## Short summary

This method sorts the data structure instantly within one call. 
It uses the passed Comparator to sort the structure or the compareTo of the contained Objects if no comparator is passed.

.. <legal notes>

legal notes
=================
| SPDX-FileCopyrightText: © 2022 ekvip automation GmbH <info@ekvip.de>
| SPDX-License-Identifier: Apache-2.0
| For details check: Apache-2.0_

.. _Apache-2.0: https://www.apache.org/licenses/LICENSE-2.0

.. </legal notes>


**Return:**``ERROR``: Sort was not able to finish 
	``SUCCESS``: Sorting was finished succesfully

*)
METHOD instantSort : CNM_CollectionInterfaces.CNM_ReturnTypes.SingleExecutionResult
VAR_INPUT
	(*The size of the list to be sorted*)
	size	: UDINT;
	(*the container, that contains the list elements*)
	container	: POINTER TO CNM_CollectionInterfaces.CNM_AbstractObject.IObject;
	(*the comparator that should be used for the sort. Must not be changed while sort is in process*)
	comparator	: CNM_CollectionInterfaces.CNM_AbstractObject.IComparator := 0;
END_VAR
VAR_IN_OUT
	(*the current version of the list, must change when the data in the list changes *)
	currentListVersion	: __XWORD;
END_VAR
VAR_INST
	cycleManager :CNM_CycleManager.SimpleCycleManager;
	index 						:__XWORD 	:=0;	
	columnindex 				:DINT;
	columnwidth 				:__XWORD;
	currentElementIndex 		:__XWORD;
	insertElementIndex 			:__XWORD;
	tmpElement 					:CNM_AbstractObject.IObject;
END_VAR
index := 0;
IF size > 1 THEN
	columnindex := THIS^.MAX_COLUMNINDEX;
	WHILE (THIS^.PREPARED_COLUMN_WIDTH[columnindex] >= size) DO
		columnindex := columnindex - 1;
	END_WHILE
	columnwidth := THIS^.PREPARED_COLUMN_WIDTH[columnindex];
	THIS^.setComparator(comparator);
ELSE
	instantSort := CNM_ReturnTypes.SingleExecutionResult.SUCCESS;
	RETURN;
END_IF

WHILE columnindex >= 0  DO  
	FOR currentElementIndex:=columnwidth TO size-1 DO
		tmpElement := container[currentElementIndex]; 
		insertElementIndex := currentElementIndex;
		WHILE 	(insertElementIndex >= columnwidth) 
			AND_THEN (THIS^.compareElements(container[insertElementIndex-columnwidth],tmpElement) = CNM_ReturnTypes.ComparationResult.GREATER)  
		DO
			container[insertElementIndex] := container[insertElementIndex-columnwidth];
			insertElementIndex := InsertElementIndex-columnwidth;
		END_WHILE
		container[insertElementIndex] := tmpElement;
	END_FOR
	columnindex := columnindex - 1;
	IF columnindex >= 0 THEN
		columnwidth := THIS^.PREPARED_COLUMN_WIDTH[columnindex];
	END_IF
END_WHILE

currentListVersion := currentListVersion + 1;
instantSort := CNM_ReturnTypes.SingleExecutionResult.SUCCESS;
END_METHOD

(*

## Short summary

This method sorts the data structure. 
It uses the passed Comperator to sort the structure.
This can take many cycles and should be called until the CNM_ReturnTypes.ExecutionState is no longer ``BUSY``.

.. <legal notes>

legal notes
=================
| SPDX-FileCopyrightText: © 2022 ekvip automation GmbH <info@ekvip.de>
| SPDX-License-Identifier: Apache-2.0
| For details check: Apache-2.0_

.. _Apache-2.0: https://www.apache.org/licenses/LICENSE-2.0

.. </legal notes>


**Return:** ``ABORTED``: While sort was pending,execute had a falling edge,
	``BUSY``: Sort is in progress
	``ERROR``: Sort was not able to finish (p.e. List changed) call sort(false) to reset
	``IDLE``: Currently no sort in progress
	``SUCCESS``: Sorting was finished 

*)
METHOD sort	:CNM_ReturnTypes.SingleExecutionState
VAR_INPUT
	(*control bit to start or abort the sorting, needs to be active until the ExecutionState is SUCCESS*)
	execute	: BOOL;
	(*The size of the list to be sorted*)
	size :UDINT;
	(*the container, that contains the list elements*)
	container	: POINTER TO CNM_AbstractObject.IObject;
	(*the comparator that should be used for the sort. Must not be changed while sort is in process*)
	comparator	: CNM_AbstractObject.IComparator	:= 0;
END_VAR
VAR_IN_OUT
	(*the current version of the list, must change when the data in the list changes *)
	currentListVersion :__XWORD;
END_VAR
VAR_INST
	cycleManager :CNM_CycleManager.SimpleCycleManager;
	index 						:__XWORD 	:=0;	
	columnindex 				:DINT 		:= 11;
	columnwidth 				:__XWORD;
	currentElementIndex 		:__XWORD;
	initCurrentElementIndex 	:__XWORD;
	insertElementIndex 			:__XWORD;
	tmpElement 					:CNM_AbstractObject.IObject;
	(* list version index, used to detect list changes during sorting *)
	lastListChangeIndex :__XWORD;
END_VAR
VAR 
	leave 						:BOOL		:= FALSE;
	operationsThisCycle 		:__XWORD	:=0;
END_VAR
VAR CONSTANT
	INIT :DINT := CNM_ReturnTypes.DefaultSteps.STEP.INIT;
	SORTING :DINT := INIT + 1;
	SUCCESS :DINT := CNM_ReturnTypes.DefaultSteps.STEP.SUCCESS;
	ERROR :DINT := CNM_ReturnTypes.DefaultSteps.STEP.ERROR;
END_VAR
cycleManager.update(execute := execute);
IF cycleManager.step.current > INIT THEN
	cycleManager.assert.bitNumber.x.valueIsEqualTo(
		currentValue := currentListVersion, 
		expectedValue := lastListChangeIndex, 
		message := 'list has changed during pending sorting'
	);
END_IF

CASE cycleManager.step.current OF
INIT:
	lastListChangeIndex := currentListVersion;
	index := 0;
	IF size > 1 THEN
		columnindex := THIS^.MAX_COLUMNINDEX;
		WHILE (THIS^.PREPARED_COLUMN_WIDTH[columnindex] >= size) DO
			columnindex := columnindex - 1;
		END_WHILE
		columnwidth := THIS^.PREPARED_COLUMN_WIDTH[columnindex];
		initCurrentElementIndex := columnwidth;
		THIS^.setComparator(comparator);
		cycleManager.proceed();
	ELSE
		cycleManager.proceedWith(SUCCESS);
	END_IF
SORTING:
	IF (lastListChangeIndex <> currentListVersion) THEN
		cycleManager.proceedWith(ERROR);
		sort := CNM_ReturnTypes.SingleExecutionState.ERROR;
		RETURN;
	END_IF
	WHILE columnindex >= 0  DO  
		FOR currentElementIndex:=initCurrentElementIndex TO size-1 DO
			tmpElement := container[currentElementIndex]; 
			insertElementIndex := currentElementIndex;
			WHILE insertElementIndex >= columnwidth  DO
				operationsThisCycle := operationsThisCycle + 1;
				IF (operationsThisCycle >= THIS^.maxCycleCompares) THEN
					leave:=TRUE;
				END_IF
				IF THIS^.compareElements(container[insertElementIndex-columnwidth],tmpElement) = CNM_ReturnTypes.ComparationResult.GREATER THEN
					container[insertElementIndex] := container[insertElementIndex-columnwidth];
					insertElementIndex := InsertElementIndex-columnwidth;
				ELSE
					EXIT;
				END_IF;
			END_WHILE
			container[insertElementIndex]:=tmpElement;
			IF leave THEN
				EXIT;
			END_IF
		END_FOR
		
		IF currentElementIndex >= size THEN
			columnindex:=columnindex-1;
			IF columnindex < 0 THEN
				lastListChangeIndex := currentListVersion := currentListVersion + 1;
				cycleManager.proceedWith(SUCCESS);
			ELSE
				columnwidth := THIS^.PREPARED_COLUMN_WIDTH[columnindex];
			END_IF
			initCurrentElementIndex := columnwidth;
		ELSE 
			initCurrentElementIndex := currentElementIndex;
			lastListChangeIndex := currentListVersion := currentListVersion + 1;
			EXIT;
		END_IF
	END_WHILE
END_CASE

sort := cycleManager.state;
END_METHOD

END_FUNCTION_BLOCK

// ---- BinaryTree/classes/BalancedBinarySearchTree.TcPOU
(*

## Short summary

Interface for a balanced, binary, search tree

- balanced means that every node has a balanced (see ``Tree_Balance``)
- binary means that every node has two childs (they can be null)
- search means it is a set, every object can be only contained once

**Attention:**
	search not only means you can't store an object with the same hash only once, instead it means you can only one element with this comparevalue.
	So if you compare elements by size and you have five diffrent objects with the same size, only one of them can be stored
	
**Warning:**
	Calling __DELETE directly on a Collection will bypass the destruct Context and therefore also delete the contained elements.
	Do not change the compare value of objects while they are in the tree, doing so will destroy your tree which can lead to not finding elements, 
	hurt of search and balanced properties and os on. If you have to alter the value the correct way is:
	remove from tree, alter, insert. Same applies for foreach / iterate do not perform any operations changing the comparevalue
	
.. <legal notes>

legal notes
=================
| SPDX-FileCopyrightText: © 2022 ekvip automation GmbH <info@ekvip.de>
| SPDX-License-Identifier: Apache-2.0
| For details check: Apache-2.0_

.. _Apache-2.0: https://www.apache.org/licenses/LICENSE-2.0

.. </legal notes>


*)

{attribute 'enable_dynamic_creation'}
FUNCTION_BLOCK BalancedBinarySearchTree EXTENDS AbstractCollection IMPLEMENTS CNM_CollectionInterfaces.IBalancedBinarySearchTree, ISetHelper, ITreeHelper
VAR
	rootNode 			:CNM_CollectionInterfaces.IBalancedBinarySearchTreeNode;
	nodeComparator		:CNM_AbstractObject.IComparator;
	(*nodestack used for iterate, placed in instance to be able to destroy it on destruct*)
	nodestack			:POINTER TO CNM_CollectionInterfaces.IBalancedBinarySearchTreeNode;
	(* set iterator for subtract *)
	subtractIterator	:CNM_CollectionInterfaces.IIterator;
	(* collection iterator for insertCollection *)
	insertIterator		:CNM_CollectionInterfaces.IIterator;
	(* set iterator for intersect *)
	intersectIterator 	:CNM_CollectionInterfaces.IIterator;
	(* the amount of compare operations per cycle *)
	upperCompareBound :UDINT := GeneralParameters.DEFAULT_OPERATIONS_PER_CYCLE;
	(* insert buffer to roll back inserted Objects in error case *)
	insertBuffer :POINTER TO CNM_AbstractObject.IObject;
	(* intersect tree *)
	intersectedTree :POINTER TO BalancedBinarySearchTree;
END_VAR

(*

## Short summary

after a double rotation balance have to be adopted

.. <legal notes>

legal notes
=================
| SPDX-FileCopyrightText: © 2022 ekvip automation GmbH <info@ekvip.de>
| SPDX-License-Identifier: Apache-2.0
| For details check: Apache-2.0_

.. _Apache-2.0: https://www.apache.org/licenses/LICENSE-2.0

.. </legal notes>



*)

METHOD PROTECTED adaptBalanceAfterDoubleRotation
VAR_INPUT
	(*the element for that childs balance should be adapted*)
	elem		:CNM_CollectionInterfaces.IBalancedBinarySearchTreeNode;
END_VAR
VAR 
	leftChild	:CNM_CollectionInterfaces.IBalancedBinarySearchTreeNode;
	rightChild	:CNM_CollectionInterfaces.IBalancedBinarySearchTreeNode;
END_VAR
__QUERYINTERFACE(elem.leftChild,leftChild);
__QUERYINTERFACE(elem.rightChild,rightChild);

CASE elem.balance OF 
	CNM_CollectionInterfaces.TreeBalance.LEFTDEEPER:
		leftChild.balance := CNM_CollectionInterfaces.TreeBalance.EQUALDEEP;
		rightChild.balance := CNM_CollectionInterfaces.TreeBalance.RIGHTDEEPER;
	CNM_CollectionInterfaces.TreeBalance.RIGHTDEEPER:
		leftChild.balance := CNM_CollectionInterfaces.TreeBalance.LEFTDEEPER;
		rightChild.balance := CNM_CollectionInterfaces.TreeBalance.EQUALDEEP;
	CNM_CollectionInterfaces.TreeBalance.EQUALDEEP:
		leftChild.balance := CNM_CollectionInterfaces.TreeBalance.EQUALDEEP;
		rightChild.balance := CNM_CollectionInterfaces.TreeBalance.EQUALDEEP;
	
END_CASE
END_METHOD


(*

## Short summary

called every time the tree changes, can be used to notify components

.. <legal notes>

legal notes
=================
| SPDX-FileCopyrightText: © 2022 ekvip automation GmbH <info@ekvip.de>
| SPDX-License-Identifier: Apache-2.0
| For details check: Apache-2.0_

.. _Apache-2.0: https://www.apache.org/licenses/LICENSE-2.0

.. </legal notes>



*)
METHOD PROTECTED announceChange
VAR_INPUT
END_VAR
THIS^.changesToCollection := THIS^.changesToCollection + 1;
END_METHOD

(*

## Short summary

check if a leftrotation is neccesary (=> is right subtree to deep?), if necessary it is performed

.. <legal notes>

legal notes
=================
| SPDX-FileCopyrightText: © 2022 ekvip automation GmbH <info@ekvip.de>
| SPDX-License-Identifier: Apache-2.0
| For details check: Apache-2.0_

.. _Apache-2.0: https://www.apache.org/licenses/LICENSE-2.0

.. </legal notes>


**Return:** returns the new root of the subtree, that replaces the node for that the rotation was checked
 
*)

METHOD PROTECTED checkLeftRotation :CNM_CollectionInterfaces.IBalancedBinarySearchTreeNode
VAR_INPUT
	(*The element for that the rotation should be checked*)
	elem				:CNM_CollectionInterfaces.IBalancedBinarySearchTreeNode;
	(*indicates if method was called in context of remove (then true) or in context of insert (then false) *)
	removing				:BOOL := FALSE;
END_VAR
VAR_IN_OUT
	(*signals if the height of any subtree has changed*)
	heightNotChanged	:BOOL;
END_VAR
IF heightNotChanged THEN 
	checkLeftRotation := elem;
	RETURN;
ELSE
	CASE elem.balance OF
		CNM_CollectionInterfaces.TreeBalance.EQUALDEEP:
			elem.balance := CNM_CollectionInterfaces.TreeBalance.RIGHTDEEPER;
			heightNotChanged := removing;
			checkLeftRotation := elem;
			RETURN;
		CNM_CollectionInterfaces.TreeBalance.LEFTDEEPER:
			elem.balance := CNM_CollectionInterfaces.TreeBalance.EQUALDEEP;
			heightNotChanged := NOT removing;
			checkLeftRotation := elem;
			RETURN;
		CNM_CollectionInterfaces.TreeBalance.RIGHTDEEPER:
			checkLeftRotation := reorganizeLeftRotate(elem := elem, heightNotChanged := heightNotChanged, removing := removing);
			RETURN;
	END_CASE
END_IF
END_METHOD

(*

## Short summary

check if a rightrotation is neccesary (=> is left subtree to deep?), if necessary it is performed

.. <legal notes>

legal notes
=================
| SPDX-FileCopyrightText: © 2022 ekvip automation GmbH <info@ekvip.de>
| SPDX-License-Identifier: Apache-2.0
| For details check: Apache-2.0_

.. _Apache-2.0: https://www.apache.org/licenses/LICENSE-2.0

.. </legal notes>


**Return:** the new root of the subtree, that replaces the node the rotation was checked for

*)

METHOD PROTECTED checkRightRotation :CNM_CollectionInterfaces.IBalancedBinarySearchTreeNode
VAR_INPUT
	(*The root of the subtree that should be checked for rotation*)
	elem 				:CNM_CollectionInterfaces.IBalancedBinarySearchTreeNode;
	(*indicates if method was called in context of remove (then true) or in context of insert (then false) *)
	removing				:BOOL	:= FALSE;
END_VAR
VAR_IN_OUT
	(*signals if the height of any subtree changed *)
	heightNotChanged 	:BOOL;
END_VAR
IF heightNotChanged THEN 
	checkRightRotation := elem;
	RETURN;
ELSE
	CASE elem.balance OF 
		CNM_CollectionInterfaces.TreeBalance.EQUALDEEP:
			elem.balance := CNM_CollectionInterfaces.TreeBalance.LEFTDEEPER;
			heightNotChanged := removing;
			checkRightRotation := elem;
			RETURN;
		CNM_CollectionInterfaces.TreeBalance.RIGHTDEEPER:
			elem.balance := CNM_CollectionInterfaces.TreeBalance.EQUALDEEP;
			heightNotChanged := NOT removing;
			checkRightRotation := elem;
			RETURN;
		CNM_CollectionInterfaces.TreeBalance.LEFTDEEPER:
			checkRightRotation := THIS^.reorganizeRightRotate(elem := elem, heightNotChanged := heightNotChanged, removing := removing);
			RETURN;
	END_CASE
END_IF
END_METHOD


(*

## Short summary

This abstract property returns the class name of the concrete object, 
which is useful to check the class name for ``__DELETE``.

.. <legal notes>

legal notes
=================
| SPDX-FileCopyrightText: © 2022 ekvip automation GmbH <info@ekvip.de>
| SPDX-License-Identifier: Apache-2.0
| For details check: Apache-2.0_

.. _Apache-2.0: https://www.apache.org/licenses/LICENSE-2.0

.. </legal notes>

*)
PROPERTY className :CNM_AbstractObject.ClassName
GET
className := 'CNM_Collections.BalancedBinarySearchTree';
END_GET
END_PROPERTY

(*

## Short summary

This method clears/deletes all clearable data from this object.

.. <legal notes>

legal notes
=================
| SPDX-FileCopyrightText: © 2022 ekvip automation GmbH <info@ekvip.de>
| SPDX-License-Identifier: Apache-2.0
| For details check: Apache-2.0_

.. _Apache-2.0: https://www.apache.org/licenses/LICENSE-2.0

.. </legal notes>



*)

METHOD clear
VAR CONSTANT
	OBJECT_NOT_REFERENCED	:__XWORD := 0;
END_VAR
THIS^.announceChange();
THIS^.destructNodeAndAllChilds(node := THIS^.rootNode, FALSE);
THIS^.rootNode := OBJECT_NOT_REFERENCED;
END_METHOD

(*

## Short summary

This method is called in the destruct method and is intended to zero all references and interfaces that should not be destructed. 
To delete the collection with all its contents, use deepDestruct() instead of destruct().

.. <legal notes>

legal notes
=================
| SPDX-FileCopyrightText: © 2025 ekvip automation GmbH <info@ekvip.de>
| SPDX-License-Identifier: Apache-2.0
| For details check: Apache-2.0_

.. _Apache-2.0: https://www.apache.org/licenses/LICENSE-2.0

.. </legal notes>

*)
METHOD PROTECTED clearContents
THIS^.clear();
THIS^.nodeComparator := 0;
END_METHOD

(*

## Short summary

This method is used to create a new instance
of the object which has the same internal state as the object.
If the object is a container class, the references to the content objects
are not cloned for this there is the method ``ICloneable.deepClone``.

If an object does not support cloning the return value is
``CNM_ReturnTypes.CloneResult.CLONE_IS_NOT_SUPPORTED``.

If there is not enough memory or the cloning fails because the
attribute enable dynamic creation was forgotten the return value is 
``CNM_ReturnTypes.CloneResult.FAILED``.

Only if the return value is ``CNM_ReturnTypes.CloneResult.SUCCESS``
the output ``clonedObject`` points to the new object
otherwise ``clonedObject`` is NULL.  

.. <legal notes>

legal notes
=================
| SPDX-FileCopyrightText: © 2022 ekvip automation GmbH <info@ekvip.de>
| SPDX-License-Identifier: Apache-2.0
| For details check: Apache-2.0_

.. _Apache-2.0: https://www.apache.org/licenses/LICENSE-2.0

.. </legal notes>


**Return:** ``CNM_ReturnTypes.CloneResult.SUCCESS``: new object clone was created,
	``CNM_ReturnTypes.CloneResult.FAILED``: object clone failed
	``CNM_ReturnTypes.CloneResult.CLONE_IS_NOT_SUPPORTED``: object does not support cloning

*)
METHOD clone :CNM_AbstractObject.CNM_ReturnTypes.CloneResult
VAR_OUTPUT
	(* new object instance or NULL if somthing went wrong *)
	clonedObject :CNM_AbstractObject.IObject;
END_VAR
VAR 
	newBalancedBinarySearchTree :POINTER TO BalancedBinarySearchTree;
	newRootObject :CNM_AbstractObject.IObject;
	newRoot : CNM_CollectionInterfaces.IBalancedBinarySearchTreeNode;
END_VAR
VAR CONSTANT
	OBJECT_NOT_REFERENCED 		:__XWORD := 0;
END_VAR
clone := THIS^.getClonedEmptyTree(deepCloned := FALSE,newBalancedBinarySearchTree => newBalancedBinarySearchTree);
clonedObject := OBJECT_NOT_REFERENCED;
IF (clone = CNM_ReturnTypes.CloneResult.SUCCESS) THEN
	IF (THIS^.size > 0) THEN
		clone := THIS^.root.clone(clonedObject => newRootObject);
		IF clone = CNM_ReturnTypes.CloneResult.SUCCESS THEN
			__QUERYINTERFACE(newRootObject,newRoot);
			newBalancedBinarySearchTree^.root := newRoot;
			newBalancedBinarySearchTree^.size := THIS^.size;
		ELSE
			newBalancedBinarySearchTree^.destruct();
			RETURN;
		END_IF	
	END_IF
	clonedObject := newBalancedBinarySearchTree^;
END_IF
END_METHOD

(*

## Short summary

compares two objects (should be nodevalues, or values to be inserted), uses the comparator set with method ``setNodeComparator``

.. <legal notes>

legal notes
=================
| SPDX-FileCopyrightText: © 2022 ekvip automation GmbH <info@ekvip.de>
| SPDX-License-Identifier: Apache-2.0
| For details check: Apache-2.0_

.. _Apache-2.0: https://www.apache.org/licenses/LICENSE-2.0

.. </legal notes>


**Return:** ``SMALLER``: ``object1`` precedes in order,
	``EQUAL``: ``object1`` and ``object2`` at the same position in order,
	``GREATER``: ``object1`` is after in order. Checkout the library CNM_ReturnTypes.

*)

METHOD PROTECTED compareNodes :CNM_ReturnTypes.ComparationResult
VAR_INPUT
	(*first object to compare*)
	object1 :CNM_AbstractObject.IObject;
	(*second object to compare*)
	object2 :CNM_AbstractObject.IObject;
END_VAR
IF THIS^.isObjectNull(THIS^.nodeComparator) THEN
	compareNodes := object1.compareTo(object2);
ELSE
	compareNodes := THIS^.nodeComparator.compare(object1,object2);
END_IF
END_METHOD


(*

## Short summary

This method compares a foreign object with the own one, this is needed for sort orders.

.. <legal notes>

legal notes
=================
| SPDX-FileCopyrightText: © 2022 ekvip automation GmbH <info@ekvip.de>
| SPDX-License-Identifier: Apache-2.0
| For details check: Apache-2.0_

.. _Apache-2.0: https://www.apache.org/licenses/LICENSE-2.0

.. </legal notes>


**Return:** ``SMALLER``: ``THIS`` precedes in order,
	``EQUAL``: ``THIS`` and ``object`` at the same position in order,
	``GREATER``: ``THIS`` is after in order.

*)
METHOD compareTo :CNM_AbstractObject.CNM_ReturnTypes.ComparationResult
VAR_INPUT
	(* foreign object to compare*)
	object	:CNM_AbstractObject.IObject;
END_VAR
VAR
	treeToCompare :POINTER TO BalancedBinarySearchTree;
END_VAR
IF THIS^.isObjectValid(object) AND_THEN __QUERYPOINTER(object,treeToCompare) THEN
	IF (THIS^.size > 0) THEN 
		compareTo := THIS^.rootNode.compareTo(treeToCompare^.root);
	ELSIF (treeToCompare^.size = 0) THEN
		compareTo := CNM_ReturnTypes.ComparationResult.EQUAL;
	ELSE
		compareTo := CNM_ReturnTypes.ComparationResult.SMALLER;
	END_IF
ELSIF THIS^.isObjectNull(object) THEN
	compareTo := CNM_ReturnTypes.ComparationResult.GREATER;
ELSE
	compareTo := CNM_ReturnTypes.ComparationResult.EQUAL;
END_IF
END_METHOD


(*

## Short summary

True if the tree contains any object where either the injected comparator or, if no comparator is used, the object.compareTo 
result is equal.

**Attention:**
	The objects can be different as long as comparesTo says they are equal, the hashcode is not considered. 
To check for same Object, use containsObject

.. <legal notes>

legal notes
=================
| SPDX-FileCopyrightText: © 2022 ekvip automation GmbH <info@ekvip.de>
| SPDX-License-Identifier: Apache-2.0
| For details check: Apache-2.0_

.. _Apache-2.0: https://www.apache.org/licenses/LICENSE-2.0

.. </legal notes>


**Return:** ``TRUE`` if an object is found for that .compareTo is equal, 
	``FALSE`` otherwise

*)

METHOD containsEqualObject :BOOL
VAR_INPUT
	(*the object to be checked if an object with equal value exists inside the collection*)
	object			:CNM_AbstractObject.IObject;
END_VAR
containsEqualObject := THIS^.getEqualObject(object);
END_METHOD


(*

## Short summary

This method checks if a given object is contained in the collection.
Overwrite default implementation to use the advantages of balanced trees

.. <legal notes>

legal notes
=================
| SPDX-FileCopyrightText: © 2022 ekvip automation GmbH <info@ekvip.de>
| SPDX-License-Identifier: Apache-2.0
| For details check: Apache-2.0_

.. _Apache-2.0: https://www.apache.org/licenses/LICENSE-2.0

.. </legal notes>


**Return:** ``FALSE``: list does not contain given object
	``TRUE``: list does contain given object

*)

METHOD containsObject :BOOL
VAR_INPUT
	(*the object to be checked if it exists inside the collection*)
	object			:CNM_AbstractObject.IObject;
END_VAR
VAR 
	currentElement	:CNM_CollectionInterfaces.IBinaryTreeNode;
END_VAR
currentElement := THIS^.rootnode;
IF THIS^.isObjectNull(currentElement) OR THIS^.isObjectNull(object) THEN
	containsObject := FALSE;
	RETURN;
END_IF
containsObject := object.isEqual(currentElement.object);
WHILE NOT containsObject DO
	CASE THIS^.compareNodes(object,currentelement.object) OF
		CNM_ReturnTypes.ComparationResult.GREATER:
			IF THIS^.isObjectValid(currentElement.rightChild) THEN 
				currentElement := currentElement.rightChild;
			ELSE	
				RETURN;
			END_IF
		CNM_ReturnTypes.ComparationResult.SMALLER:
			IF THIS^.isObjectValid(currentElement.leftChild) THEN
				currentElement := currentElement.leftChild;
			ELSE
				RETURN;
			END_IF
		ELSE
			// if reached, the node comparator founds both objects equal but object.isEqual not
			RETURN;
	END_CASE
	containsObject := object.isEqual(currentElement.object);
END_WHILE
END_METHOD

(*

## Short summary

This method returns a NEW Iterator instance which can iterate the collection.
These iterators can be used parallel independend of each other on the same collection.

**Warning:**
The returned Iterator was created using the __NEW operator and must be destructed to avoid memory leaks!



.. <legal notes>

legal notes
=================
| SPDX-FileCopyrightText: © 2024 ekvip automation GmbH <info@ekvip.de>
| SPDX-License-Identifier: Apache-2.0
| For details check: Apache-2.0_

.. _Apache-2.0: https://www.apache.org/licenses/LICENSE-2.0

.. </legal notes>



*)
METHOD createNewIterator : CNM_CollectionInterfaces.CNM_ReturnTypes.SingleExecutionResult
VAR_OUTPUT
	(*The new created iterator or null if allocation fails *)
	iterator	: CNM_CollectionInterfaces.IIterator;
END_VAR
VAR
	newIterator :POINTER TO InorderBBSTIterator;
END_VAR
newIterator := __NEW(InorderBBSTIterator(tree := THIS^));
IF (newIterator = 0) THEN
	createNewIterator := CNM_ReturnTypes.SingleExecutionResult.ERROR;
	RETURN;
END_IF
createNewIterator := CNM_ReturnTypes.SingleExecutionResult.SUCCESS;
__QUERYINTERFACE(newIterator^, iterator);
END_METHOD

(*

## Short summary

Method to decrease \_\_XWORD without overflow

.. <legal notes>

legal notes
=================
| SPDX-FileCopyrightText: © 2022 ekvip automation GmbH <info@ekvip.de>
| SPDX-License-Identifier: Apache-2.0
| For details check: Apache-2.0_

.. _Apache-2.0: https://www.apache.org/licenses/LICENSE-2.0

.. </legal notes>



*)
METHOD PRIVATE dec
VAR_IN_OUT
	(*value to decrease*)
	value 		:__XWORD;
END_VAR
value := SEL(value = 0, value - 1 , 0);
END_METHOD

(*

## Short summary

decrements the size of the collection

.. <legal notes>

legal notes
=================
| SPDX-FileCopyrightText: © 2022 ekvip automation GmbH <info@ekvip.de>
| SPDX-License-Identifier: Apache-2.0
| For details check: Apache-2.0_

.. _Apache-2.0: https://www.apache.org/licenses/LICENSE-2.0

.. </legal notes>



*)

METHOD PROTECTED decrementSize
VAR_INPUT
END_VAR
THIS^.collectionSize := THIS^.collectionSize-1;
END_METHOD

(*

## Short summary

This method is used to create a new instance
of the object which has the same internal state as the object.
If the object is a container class, the references to the content objects
are cloned too.

If an object does not support cloning the return value is
``CNM_ReturnTypes.CloneResult.CLONE_IS_NOT_SUPPORTED``.

If there is not enough memory or the cloning fails because the
attribute enable dynamic creation was forgotten the return value is 
``CNM_ReturnTypes.CloneResult.FAILED``.
If something goes wrong, then this method must clean up everything
that has been cloned and free the memory again.
**The deepClone either works completely, or not at all**

Only if the return value is ``CNM_ReturnTypes.CloneResult.SUCCESS``
the output ``clonedObject`` points to the new object
otherwise ``clonedObject`` is NULL.  

.. <legal notes>

legal notes
=================
| SPDX-FileCopyrightText: © 2022 ekvip automation GmbH <info@ekvip.de>
| SPDX-License-Identifier: Apache-2.0
| For details check: Apache-2.0_

.. _Apache-2.0: https://www.apache.org/licenses/LICENSE-2.0

.. </legal notes>


**Return:** ``CNM_ReturnTypes.CloneResult.SUCCESS``: new object clone was created,
	``CNM_ReturnTypes.CloneResult.FAILED``: object clone failed
	``CNM_ReturnTypes.CloneResult.CLONE_IS_NOT_SUPPORTED``: object does not support deep cloning

*)
METHOD deepClone :CNM_ReturnTypes.CloneResult
VAR_OUTPUT
	(* new object instance or NULL if somthing went wrong *)
	clonedObject	:CNM_AbstractObject.IObject;
END_VAR
VAR
	newTreeObject 	:CNM_AbstractObject.IObject;
	newTree 		:POINTER TO BalancedBinarySearchTree;
	currentNode 	:CNM_CollectionInterfaces.IBalancedBinarySearchTreeNode;
	binaryRoot 		:CNM_CollectionInterfaces.IBalancedBinarySearchTreeNode;
	rootObject		:CNM_AbstractObject.IObject;
END_VAR
clonedObject := 0;

deepClone := THIS^.getClonedEmptyTree(
	deepCloned := TRUE, 
	newBalancedBinarySearchTree => newTree
);

RETURN (deepClone <> CNM_ReturnTypes.CloneResult.SUCCESS);
clonedObject := newTree^;
RETURN (THIS^.size = 0);
deepClone := THIS^.root.deepClone(clonedObject => rootObject);

IF ((deepClone = CNM_ReturnTypes.CloneResult.SUCCESS) AND_THEN THIS^.isObjectValid(rootObject)) THEN
	__QUERYINTERFACE(rootObject,binaryRoot);
	newTree^.root := binaryRoot;
	newTree^.size := THIS^.size;
ELSE
	newTree^.deepDestruct();
END_IF
END_METHOD

(*

## Short summary

destructs / deepdestructs all nodes in the subtrees of a specified node and this node

.. <legal notes>

legal notes
=================
| SPDX-FileCopyrightText: © 2022 ekvip automation GmbH <info@ekvip.de>
| SPDX-License-Identifier: Apache-2.0
| For details check: Apache-2.0_

.. _Apache-2.0: https://www.apache.org/licenses/LICENSE-2.0

.. </legal notes>



*)

METHOD PROTECTED destructNodeAndAllChilds
VAR_INPUT
	(*the node that should be destructed with all it's childs*)
	node							:CNM_CollectionInterfaces.IBinaryTreeNode;
END_VAR
VAR_INPUT
	(*if true also the node contents will be destructed, if false only the nodes will be destructed*)
	destructNodeContents			:BOOL;
END_VAR
VAR
	child 							:CNM_CollectionInterfaces.IBinaryTreeNode;
END_VAR
VAR CONSTANT
	OBJECT_NOT_REFERENCED			:__XWORD := 0;
END_VAR
IF THIS^.isObjectNull(node) THEN
    RETURN;
END_IF

IF THIS^.isObjectValid(node.leftChild) THEN
	child := node.leftChild;
	THIS^.destructNodeAndAllChilds(node := child, destructNodeContents := destructNodeContents);
	node.leftChild := OBJECT_NOT_REFERENCED;
END_IF
IF THIS^.isObjectValid(node.rightChild) THEN
	child := node.rightChild;
	THIS^.destructNodeAndAllChilds(node := child, destructNodeContents := destructNodeContents);
	node.rightChild := OBJECT_NOT_REFERENCED;
END_IF
IF destructNodeContents THEN
	node.deepDestruct();
ELSE
	node.destruct();	
END_IF
THIS^.decrementSize();
END_METHOD

(*

## Short summary

Mark the object as deleted, as it stays in the memory.

.. <legal notes>

legal notes
=================
| SPDX-FileCopyrightText: © 2022 ekvip automation GmbH <info@ekvip.de>
| SPDX-License-Identifier: Apache-2.0
| For details check: Apache-2.0_

.. _Apache-2.0: https://www.apache.org/licenses/LICENSE-2.0

.. </legal notes>

*)
METHOD FB_Exit : BOOL
VAR_INPUT
	(* TRUE: the exit method is called in order to leave the instance which will be copied afterwards (online change).*)
	bInCopyCode	: BOOL;
END_VAR
IF 
	THIS^.isObjectValid(THIS^.rootNode) 
THEN	
	THIS^.destructNodeAndAllChilds(node := THIS^.rootNode, destructNodeContents := TRUE);
END_IF
IF THIS^.isObjectValid(THIS^.nodeComparator) THEN
	THIS^.nodeComparator.deepDestruct();
END_IF
IF (THIS^.nodestack <> 0) THEN
	__DELETE(THIS^.nodestack);
END_IF
IF THIS^.isObjectValid(THIS^.subtractIterator) THEN
	THIS^.subtractIterator.deepDestruct();
END_IF
IF THIS^.isObjectValid(THIS^.insertIterator) THEN
	THIS^.insertIterator.deepDestruct();
END_IF
IF THIS^.isObjectValid(THIS^.intersectIterator) THEN
	THIS^.intersectIterator.deepDestruct();
END_IF
IF THIS^.insertBuffer <> 0 THEN
	__DELETE(THIS^.insertBuffer);
END_IF
IF THIS^.intersectedTree <> 0 THEN
	__DELETE(THIS^.intersectedTree);
END_IF
END_METHOD

(*

## Short summary

The constructor ``FB_init`` is needed to create an unique hash code.
The hash code is a pseudo random number create with a [xorshift](https://en.wikipedia.org/wiki/Xorshift) algorithm.
It can be overwritten on derivations, because it will be called implicit, ``SUPER^.FB_init()`` is not required.
For more information check: [Behavoir with derived function blocks](https://infosys.beckhoff.com/content/1033/tc3_plc_intro/5482088715.html?id=6983869892358031022).

.. <legal notes>

legal notes
=================
| SPDX-FileCopyrightText: © 2022 ekvip automation GmbH <info@ekvip.de>
| SPDX-License-Identifier: Apache-2.0
| For details check: Apache-2.0_

.. _Apache-2.0: https://www.apache.org/licenses/LICENSE-2.0

.. </legal notes>



*)

METHOD FB_init : BOOL
VAR_INPUT
	(* if TRUE, the retain variables are initialized (warm start / cold start)*)
	bInitRetains	:BOOL;
	(* if TRUE, the instance afterwards gets moved into the copy code (online change) *)
	bInCopyCode		:BOOL;  
	(*Optional comparator*)
	nodeComparator 	:CNM_AbstractObject.IComparator	:= OBJECT_NOT_REFERENCED;
END_VAR
VAR
	{attribute 'hide'}
	newHashstate3		:CNM_AbstractObject.Hashcode;
END_VAR
VAR CONSTANT
	{attribute 'hide'}
	NUMBER_OF_LEFT_SHIFTS		:UINT	:= 17;
	{attribute 'hide'}
	NUMBER_OF_LEFT_ROTATIONS	:UINT   := 45;
	OBJECT_NOT_REFERENCED 		:__XWORD := 0;
END_VAR
THIS^.collectionSize := 0;
THIS^.nodeComparator := nodeComparator;
END_METHOD

(*

## Short summary

prepares a new Comparator (if set)

.. <legal notes>

legal notes
=================
| SPDX-FileCopyrightText: © 2022 ekvip automation GmbH <info@ekvip.de>
| SPDX-License-Identifier: Apache-2.0
| For details check: Apache-2.0_

.. _Apache-2.0: https://www.apache.org/licenses/LICENSE-2.0

.. </legal notes>



*)

METHOD PROTECTED getClonedComparator : CNM_ReturnTypes.CloneResult
VAR_INPUT
	(*True if called from deepclonecontext*)
	deepCloned :BOOL;
END_VAR
VAR
	newComparatorObject 		:CNM_AbstractObject.IObject;
END_VAR
VAR_OUTPUT
	(*New comparator Object, null if not existent or not cloneable*)
	newComparator 				:CNM_AbstractObject.IComparator;
END_VAR
IF deepCloned THEN
	IF NOT	(((
				getClonedComparator := THIS^.nodeComparator.deepClone(clonedObject => newComparatorObject)
			) = (	
				CNM_ReturnTypes.CloneResult.SUCCESS
			)
		) AND_THEN (
			__QUERYINTERFACE(newComparatorObject, newComparator)
		)
	) THEN
		getClonedComparator := CNM_ReturnTypes.CloneResult.FAILED;
		IF THIS^.isObjectValid(newComparatorObject) THEN
			newComparatorObject.deepDestruct();
		END_IF;		
		RETURN;	
	END_IF
ELSE
	IF NOT	(((
				getClonedComparator := THIS^.nodeComparator.clone(clonedObject => newComparatorObject)
			) = (	
				CNM_ReturnTypes.CloneResult.SUCCESS
			)
		) AND_THEN (
			__QUERYINTERFACE(newComparatorObject, newComparator)
		)
	) THEN
		getClonedComparator := CNM_ReturnTypes.CloneResult.FAILED;
		IF THIS^.isObjectValid(newComparatorObject) THEN
			newComparatorObject.destruct();
		END_IF;		
		RETURN;	
	END_IF
END_IF
END_METHOD

(*

## Short summary

prepares a new empty tree object with the same internal state as THIS^

.. <legal notes>

legal notes
=================
| SPDX-FileCopyrightText: © 2022 ekvip automation GmbH <info@ekvip.de>
| SPDX-License-Identifier: Apache-2.0
| For details check: Apache-2.0_

.. _Apache-2.0: https://www.apache.org/licenses/LICENSE-2.0

.. </legal notes>



*)

METHOD PROTECTED getClonedEmptyTree :CNM_ReturnTypes.CloneResult;
VAR_INPUT
	(*indicates if tree should be cloned or deepcloned*)
	deepCloned					:BOOL;
END_VAR
VAR_OUTPUT
	newBalancedBinarySearchTree :POINTER TO BalancedBinarySearchTree;
END_VAR
VAR
	comparator 					: CNM_AbstractObject.IComparator;
END_VAR
VAR CONSTANT
	OBJECT_NOT_REFERENCED 		:__XWORD := 0;
END_VAR
getClonedEmptyTree := CNM_ReturnTypes.CloneResult.SUCCESS;
IF 	THIS^.isObjectValid(THIS^.nodeComparator) THEN
	getClonedEmptyTree := getClonedComparator(deepCloned := deepCloned, newComparator => comparator);
END_IF;
IF getClonedEmptyTree = CNM_ReturnTypes.CloneResult.SUCCESS THEN
	newBalancedBinarySearchTree := __NEW(
	BalancedBinarySearchTree(nodeComparator := comparator)
	);
	getClonedEmptyTree := CNM_AbstractObject.CNM_ReturnTypes.CloneResult.SUCCESS;
END_IF
END_METHOD

(*

## Short summary

Searches an Object, that is equal to the provided object in terms of the compareTo Method (or an provided comparator from the parentstructure). 
Does not care about equal or not equal hashcodes.
 
.. <legal notes>

legal notes
=================
| SPDX-FileCopyrightText: © 2023 ekvip automation GmbH <info@ekvip.de>
| SPDX-License-Identifier: Apache-2.0
| For details check: Apache-2.0_

.. _Apache-2.0: https://www.apache.org/licenses/LICENSE-2.0

.. </legal notes>


**Return:** True when an object that is equal is found, false else

*)

METHOD INTERNAL getEqualObject :BOOL
VAR_INPUT
	(*The object for that an aquvivelent is searched*)
	object :CNM_AbstractObject.IObject;
END_VAR
VAR_OUTPUT
	(*The found object or null if not found*)
	foundObject :CNM_AbstractObject.IObject;
END_VAR
VAR 
	currentNode 			:CNM_CollectionInterfaces.IBinaryTreeNode;
END_VAR
VAR CONSTANT
	OBJECT_NOT_REFERENCED 	:__XWORD := 0;
END_VAR
currentNode := THIS^.rootNode;
getEqualObject := FALSE;
foundObject := OBJECT_NOT_REFERENCED;

IF THIS^.isObjectNull(currentNode) OR_ELSE THIS^.isObjectNull(object) THEN
	getEqualObject := FALSE;
	RETURN;
END_IF
WHILE THIS^.isObjectValid(currentNode) DO
	CASE THIS^.compareNodes(object1 := object, object2 := currentNode.object) OF
		CNM_ReturnTypes.ComparationResult.EQUAL:
			foundObject := currentNode.object;
			getEqualObject := TRUE;
			RETURN;
		CNM_ReturnTypes.ComparationResult.SMALLER:
			currentNode := currentNode.leftChild;
		CNM_ReturnTypes.ComparationResult.GREATER:
			currentNode := currentNode.rightChild;
	END_CASE
END_WHILE
END_METHOD

(*

## Short summary

finds the next greater node (inorder successor) of a specified node
 
.. <legal notes>

legal notes
=================
| SPDX-FileCopyrightText: © 2022 ekvip automation GmbH <info@ekvip.de>
| SPDX-License-Identifier: Apache-2.0
| For details check: Apache-2.0_

.. _Apache-2.0: https://www.apache.org/licenses/LICENSE-2.0

.. </legal notes>


**Return:** ``TRUE`` if inorder successor is found, ``FALSE`` else

*)

METHOD PROTECTED getInorderSuccessor :BOOL

VAR_IN_OUT
	nodebuffer				:POINTER TO CNM_CollectionInterfaces.IBinaryTreeNode;
	bufferindex				:__XWORD;
END_VAR
VAR_OUTPUT
	(*if successor is found then successor, else null*)
	successor				:CNM_CollectionInterfaces.IBinaryTreeNode;
END_VAR
VAR_INST
	currentNode 		:CNM_CollectionInterfaces.IBinaryTreeNode;
END_VAR
VAR CONSTANT 
	OBJECT_NOT_REFERENCED	:__XWORD := 0;
END_VAR
IF THIS^.isObjectNull(currentNode) THEN
	currentNode := nodebuffer[bufferindex];
	nodebuffer[bufferindex] := OBJECT_NOT_REFERENCED;
	dec(bufferindex);
END_IF
successor := currentNode;
getInorderSuccessor := THIS^.isObjectValid(currentNode) OR THIS^.isObjectValid(nodebuffer[bufferindex]);
IF THIS^.isObjectValid(currentNode) THEN
	currentNode := THIS^.getSmallestNode(startNode := currentNode.rightChild,nodebuffer := nodebuffer, bufferindex := bufferindex);	
END_IF
END_METHOD

(*

## Short summary

finds the smallest node in a specified (sub)tree

.. <legal notes>

legal notes
=================
| SPDX-FileCopyrightText: © 2022 ekvip automation GmbH <info@ekvip.de>
| SPDX-License-Identifier: Apache-2.0
| For details check: Apache-2.0_

.. _Apache-2.0: https://www.apache.org/licenses/LICENSE-2.0

.. </legal notes>


**Return:** the node with the smallest value based on the comparedTo Method

*)

METHOD PROTECTED getSmallestNode :CNM_CollectionInterfaces.IBinaryTreeNode
VAR_INPUT
	(*the node from that the search should be started*)
	startNode 				:CNM_CollectionInterfaces.IBinaryTreeNode;
END_VAR
VAR_IN_OUT
	nodebuffer				:POINTER TO CNM_CollectionInterfaces.IBinaryTreeNode;
	bufferindex				:__XWORD;
END_VAR
VAR
	currNode				:CNM_CollectionInterfaces.IBinaryTreeNode;
END_VAR
VAR CONSTANT 
	OBJECT_NOT_REFERENCED	:__XWORD := 0;
END_VAR
IF THIS^.isObjectValid(startNode) THEN
	currNode := startNode;
	IF THIS^.isObjectValid(startNode.leftChild) THEN
		IF THIS^.isObjectValid(nodebuffer[bufferindex]) THEN
			inc(bufferindex);
		END_IF
		nodebuffer[bufferindex] := currNode;
		inc(bufferindex);
		currNode := currNode.leftChild;
	ELSE
		getSmallestNode := startNode;
		RETURN;
	END_IF
	WHILE THIS^.isObjectValid(currNode.leftChild) DO		
		nodebuffer[bufferindex] := currNode;
		currNode := currNode.leftChild;
		inc(bufferindex);
	END_WHILE
	dec(bufferindex);
	getSmallestNode := currNode;
	RETURN;
ELSE
	getSmallestNode := OBJECT_NOT_REFERENCED;
END_IF
END_METHOD

(*

## Short summary

method to increase \_\_xword without overflow

.. <legal notes>

legal notes
=================
| SPDX-FileCopyrightText: © 2022 ekvip automation GmbH <info@ekvip.de>
| SPDX-License-Identifier: Apache-2.0
| For details check: Apache-2.0_

.. _Apache-2.0: https://www.apache.org/licenses/LICENSE-2.0

.. </legal notes>



*)
METHOD PRIVATE inc
VAR_IN_OUT
	value 		:__XWORD;
END_VAR
VAR CONSTANT
	XWORD_MAX	:__XWORD 	:= TO___XWORD(0 - 1);
END_VAR
value := SEL(value = XWORD_MAX, value + 1, XWORD_MAX);
END_METHOD

(*

## Short summary

increments the size of the collection

.. <legal notes>

legal notes
=================
| SPDX-FileCopyrightText: © 2022 ekvip automation GmbH <info@ekvip.de>
| SPDX-License-Identifier: Apache-2.0
| For details check: Apache-2.0_

.. _Apache-2.0: https://www.apache.org/licenses/LICENSE-2.0

.. </legal notes>



*)


METHOD PROTECTED incrementSize
VAR_INPUT
END_VAR
THIS^.collectionSize := THIS^.collectionSize+1;
END_METHOD


(*

## Short summary

This method can be used to insert a single element into the tree.
It will only be inserted if the tree does not already contain an equal element.

.. <legal notes>

legal notes
=================
| SPDX-FileCopyrightText: © 2022 ekvip automation GmbH <info@ekvip.de>
| SPDX-License-Identifier: Apache-2.0
| For details check: Apache-2.0_

.. _Apache-2.0: https://www.apache.org/licenses/LICENSE-2.0

.. </legal notes>


**Return:** ``SUCCESS``: operation successful
	``ABORTED``: object was already contained, null object was passed or the tree itself was passed
	``ERROR``: container allocation failed or tree itself was inconsistent
*)

METHOD INTERNAL insert :CNM_ReturnTypes.SingleExecutionResult
VAR_INPUT
	(*The object that should be inserted*)
	object				:CNM_AbstractObject.IObject;
END_VAR
VAR 
	heightNotChanged	:BOOL	:= TRUE;
	returnedRoot 		:CNM_CollectionInterfaces.IBalancedBinarySearchTreeNode;
END_VAR
insert := CNM_ReturnTypes.SingleExecutionResult.ABORTED;
RETURN(THIS^.isObjectNull(object) OR_ELSE THIS^.isEqual(object));

returnedRoot := THIS^.recursivInsert(
	object := object,
	elem := THIS^.rootNode,
	heightNotChanged := heightNotChanged,
	insertResult => insert
);

IF insert = CNM_ReturnTypes.SingleExecutionResult.SUCCESS THEN
	THIS^.rootNode := returnedRoot;
	THIS^.announceChange();
	THIS^.incrementSize();
END_IF
END_METHOD

(*

## Short summary

This method inserts all elements of a collection into the tree.

If any value of the collection could not be inserted because of duplication, operation isn't aborted, 
insertion is tried for every element of the collection.

.. <legal notes>

legal notes
=================
| SPDX-FileCopyrightText: © 2025 ekvip automation GmbH <info@ekvip.de>
| SPDX-License-Identifier: Apache-2.0
| For details check: Apache-2.0_

.. _Apache-2.0: https://www.apache.org/licenses/LICENSE-2.0

.. </legal notes>


**Return:** ``SUCCESS``: if insert could be made
	``ABORTED``: execute has a falling edge during insert,
	``BUSY``: Insert is in Progress
	``ERROR``: the passed collection where not valid / contained invalid Elements
	``IDLE``: method was never started

*)
METHOD INTERNAL insertCollection :CNM_ReturnTypes.SingleExecutionState
VAR_INPUT
	(*The collection that should be inserted*)
	collection					:CNM_CollectionInterfaces.ICollection;
	(*If insert should be processed*)
	execute 					:BOOL;
END_VAR
VAR_INST
	cycleManager		:CNM_CycleManager.SimpleCycleManager;
	index :LINT := 0;
	insertFailed :BOOL;
END_VAR
VAR
	iterateObject 				:CNM_AbstractObject.IObject;
	insertOperationsThisCycle	:__XWORD := 0;
END_VAR
VAR CONSTANT
	INIT :DINT := CNM_ReturnTypes.DefaultSteps.STEP.INIT;
	PROCESSING :DINT := INIT + 1;
	ROLL_BACK :DINT := PROCESSING + 1;
	CLEAN_UP :DINT := ROLL_BACK + 1;
	SUCCESS :DINT := CNM_ReturnTypes.DefaultSteps.STEP.SUCCESS;
	ERROR :DINT := CNM_ReturnTypes.DefaultSteps.STEP.ERROR;
END_VAR
REPEAT
	cycleManager(execute := execute);
	CASE cycleManager.step.current OF
	INIT:
		insertFailed := FALSE;
		cycleManager.configuration.sequence.requireSuccessStep := FALSE;
		IF THIS^.isObjectNull(collection) OR_ELSE THIS^.isEqual(collection) THEN
			cycleManager.proceedWith(ERROR);
			CONTINUE;
		END_IF
		IF collection.isEmpty THEN
			cycleManager.proceedWith(SUCCESS);
			CONTINUE;
		END_IF
		IF THIS^.insertBuffer <> 0 THEN
			__DELETE(THIS^.insertBuffer);
		END_IF
		THIS^.insertBuffer := __NEW(__XWORD, collection.size);
		IF THIS^.isObjectValid(THIS^.insertIterator) THEN
			THIS^.insertIterator.destruct();
		END_IF
		IF (collection.createNewIterator(iterator => THIS^.insertIterator) <> CNM_ReturnTypes.SingleExecutionResult.SUCCESS)
		THEN
			cycleManager.proceedWith(ERROR);
			CONTINUE;
		END_IF
		THIS^.insertIterator.iterate(execute := FALSE);
		index := 0;
		cycleManager.proceed();
	
	PROCESSING:
		WHILE 	(insertOperationsThisCycle < THIS^.maxCycleCompares) DO
			CASE THIS^.insertIterator.iterate(execute := TRUE, object => iterateObject) OF
			CNM_ReturnTypes.SingleExecutionState.BUSY:
				CASE THIS^.insert(object := iterateObject) OF
				CNM_ReturnTypes.SingleExecutionResult.ERROR:
					cycleManager.proceedWith(ROLL_BACK);
					EXIT;
				CNM_ReturnTypes.SingleExecutionResult.SUCCESS:
					THIS^.insertBuffer[index] := iterateObject;
					index := index + 1;
				END_CASE
				insertOperationsThisCycle := (insertOperationsThisCycle + THIS^.treeHeight);
				
			CNM_ReturnTypes.SingleExecutionState.SUCCESS:
				cycleManager.proceedWith(CLEAN_UP);
				EXIT;
			ELSE
				cycleManager.proceedWith(ROLL_BACK);
				EXIT;
			END_CASE
		END_WHILE
	ROLL_BACK:
		insertFailed := TRUE;
		REPEAT 
			THIS^.remove(THIS^.insertBuffer[index]);
			index := index - 1;
		UNTIL
			(index < 0)
		END_REPEAT 
		cycleManager.proceed();
	CLEAN_UP:
		__DELETE(THIS^.insertBuffer);
		IF THIS^.isObjectValid(THIS^.insertIterator) THEN
			THIS^.insertIterator.destruct();
			THIS^.insertIterator := 0;
		END_IF
		cycleManager.proceedWith(
			step := SEL(insertFailed, SUCCESS, ERROR)
		);  
	END_CASE
UNTIL 
	(
		(cycleManager.state <> CNM_ReturnTypes.SingleExecutionState.BUSY) 
	OR_ELSE
		(insertOperationsThisCycle >= THIS^.maxCycleCompares)
	)
END_REPEAT

insertCollection := cycleManager.state;
END_METHOD

(*

## Short summary

This method inserts all elements of a collection into the tree
This takes only one cycle.

.. <legal notes>

legal notes
=================
| SPDX-FileCopyrightText: © 2022 ekvip automation GmbH <info@ekvip.de>
| SPDX-License-Identifier: Apache-2.0
| For details check: Apache-2.0_

.. _Apache-2.0: https://www.apache.org/licenses/LICENSE-2.0

.. </legal notes>


**Return:** ``SingleExecutionResult.SUCCESS``: operation successful
	``SingleExecutionResult.ERROR``: out of memory
	``SingleExecutionResult.ABORTED``: collection to insert wasn't valid (NULL) or the tree itself was passed

*)
METHOD INTERNAL instantInsertCollection : CNM_ReturnTypes.SingleExecutionResult
VAR_INPUT
	(*The collection that should be inserted*) 
	collection	: CNM_CollectionInterfaces.ICollection;
END_VAR
VAR
	insertIterator :CNM_CollectionInterfaces.IIterator;
	insertObject :CNM_AbstractObject.IObject;
	insertedObjects :POINTER TO CNM_AbstractObject.IObject;
	index :LINT := 0;
	iteratorState :CNM_ReturnTypes.SingleExecutionState;
	insertWasError :BOOL := FALSE;
END_VAR
VAR CONSTANT
	NULL :__XWORD := 0;
END_VAR
instantInsertCollection := CNM_ReturnTypes.SingleExecutionResult.ABORTED;
RETURN( THIS^.isObjectNull(collection) OR_ELSE THIS^.isEqual(collection));
IF collection.isEmpty THEN
	instantInsertCollection := CNM_ReturnTypes.SingleExecutionResult.SUCCESS;
	RETURN;
END_IF

insertedObjects := __NEW(__XWORD, collection.size);
IF insertedObjects = NULL THEN
	instantInsertCollection := CNM_ReturnTypes.SingleExecutionResult.ERROR;
	RETURN;
END_IF

IF (collection.createNewIterator(iterator => insertIterator) 
 <> CNM_ReturnTypes.SingleExecutionResult.SUCCESS)
THEN
	IF insertIterator <> 0 THEN
		insertIterator.destruct();
	END_IF
	__DELETE(insertedObjects); 
 	instantInsertCollection := CNM_ReturnTypes.SingleExecutionResult.ERROR;
END_IF
instantInsertCollection := CNM_ReturnTypes.SingleExecutionResult.SUCCESS;
insertIterator.iterate(execute := FALSE);
WHILE (
	(iteratorstate := insertIterator.iterate(execute := TRUE, object => insertObject)) 
 	= CNM_ReturnTypes.SingleExecutionState.BUSY
) DO
	CASE THIS^.insert(insertObject) OF
	CNM_ReturnTypes.SingleExecutionResult.SUCCESS:
		insertedObjects[index] := insertObject;
		index := index +1;
	CNM_ReturnTypes.SingleExecutionResult.ERROR: 
		insertWasError := TRUE;
		EXIT;
	END_CASE
END_WHILE

IF insertWasError OR_ELSE (iteratorState <> CNM_ReturnTypes.SingleExecutionState.SUCCESS) THEN
	REPEAT 
		THIS^.remove(insertedObjects[index]);
		index := index - 1;
	UNTIL
		(index < 0)
	END_REPEAT 
	instantInsertCollection := CNM_ReturnTypes.SingleExecutionResult.ERROR;
END_IF

__DELETE(insertedObjects);
insertIterator.destruct();
END_METHOD

(*

## Short summary

overwrites the content of this set with the intersection of this set and the given set
Set intersection: Common elements between two sets.

**Example:**
Set A = {2, 3, 1, 4}
Set B = {3, 5, 6, 4}

Intersection of A and B: {3, 4}

.. <legal notes>

legal notes
=================
| SPDX-FileCopyrightText: © 2022 ekvip automation GmbH <info@ekvip.de>
| SPDX-License-Identifier: Apache-2.0
| For details check: Apache-2.0_

.. _Apache-2.0: https://www.apache.org/licenses/LICENSE-2.0

.. </legal notes>


**Return:** ``SingleExecutionResult.SUCCESS``: if intersect is complete
	``SingleExecutionResult.ABORTED``: foreign set wasn't valid

*)
METHOD INTERNAL instantIntersect : CNM_ReturnTypes.SingleExecutionResult
VAR_INPUT
	(*foreign set to intersect with*)
	set	: CNM_CollectionInterfaces.ISet;
END_VAR
VAR
	iteratorState :CNM_ReturnTypes.SingleExecutionState;
	iterator :CNM_CollectionInterfaces.IIterator;
	newTree :BalancedBinarySearchTree(THIS^.nodeComparator);
	iteratedObject :CNM_AbstractObject.IObject;
	equalObject :CNM_AbstractObject.IObject;
END_VAR
instantIntersect := CNM_ReturnTypes.SingleExecutionResult.ABORTED;
RETURN(THIS^.isObjectNull(set) OR_ELSE THIS^.isEqual(set));
IF set.size = 0 THEN
	THIS^.clear();
	instantIntersect := CNM_ReturnTypes.SingleExecutionResult.SUCCESS;
	RETURN;
END_IF

IF (set.createNewIterator(iterator => iterator)
 <> CNM_ReturnTypes.SingleExecutionResult.SUCCESS)
THEN
	IF iterator <> 0 THEN
		iterator.destruct();
	END_IF
	newTree.destruct();
 	instantIntersect := CNM_ReturnTypes.SingleExecutionResult.ERROR;
END_IF

iterator.iterate(execute := FALSE);
REPEAT 
	iteratorState := iterator.iterate(execute := TRUE, object => iteratedObject); 
	CASE iteratorState OF
	CNM_ReturnTypes.SingleExecutionState.BUSY:
		IF THIS^.getEqualObject(object := iteratedObject, foundObject => equalObject) THEN
			IF (newTree.insert(equalObject) = CNM_ReturnTypes.SingleExecutionResult.ERROR) THEN
				iterator.destruct();
				newTree.destruct();
				instantIntersect := CNM_ReturnTypes.SingleExecutionResult.ERROR;
				RETURN;
			END_IF
		END_IF
		
	CNM_ReturnTypes.SingleExecutionState.ERROR:
		iterator.destruct();
		newTree.destruct();
		instantIntersect := CNM_ReturnTypes.SingleExecutionResult.ERROR;
		RETURN;
	END_CASE
UNTIL
	(iteratorState = CNM_ReturnTypes.SingleExecutionState.SUCCESS)
END_REPEAT

THIS^.clear();
THIS^.root := newTree.root;
THIS^.size := newTree.size;
newTree.root := 0;
newTree.destruct();
iterator.destruct();
END_METHOD

(*

## Short summary

overwrites the content of this set with the union of this set and the given set
Set union: Combination of all elements from two sets.

**Example:**
Set A = {2, 3, 1, 4}
Set B = {3, 5, 6, 4}

Union of A and B: {1, 2, 3, 4, 5, 6}

.. <legal notes>

legal notes
=================
| SPDX-FileCopyrightText: © 2022 ekvip automation GmbH <info@ekvip.de>
| SPDX-License-Identifier: Apache-2.0
| For details check: Apache-2.0_

.. _Apache-2.0: https://www.apache.org/licenses/LICENSE-2.0

.. </legal notes>


**Return:** ``SUCCESS``: if merge completed
	```SingleExecutionResult.ABORTED``: foreign set wasn't valid

*)
METHOD INTERNAL instantMerge : CNM_ReturnTypes.SingleExecutionResult
VAR_INPUT
	(*foreign set to merge with*)
	set	: CNM_CollectionInterfaces.ISet;
END_VAR
instantMerge := THIS^.instantInsertCollection(collection := set);
END_METHOD

(*

## Short summary

overwrites the content of this set with the set difference of this set and the given set
Set difference: Elements present in one set but not in the other.

**Example:**
Set A = {2, 3, 1, 4}
Set B = {3, 5, 6, 4}

Set difference (A - B): {1, 2}
Set difference (B - A): {5, 6}

.. <legal notes>

legal notes
=================
| SPDX-FileCopyrightText: © 2022 ekvip automation GmbH <info@ekvip.de>
| SPDX-License-Identifier: Apache-2.0
| For details check: Apache-2.0_

.. _Apache-2.0: https://www.apache.org/licenses/LICENSE-2.0

.. </legal notes>


**Return:** ``SingleExecutionResult.SUCCESS``: if insert could made, error if object was already in the tree,
	```SingleExecutionResult.ABORTED``: foreign set wasn't valid

*)
METHOD INTERNAL instantSubtract : CNM_ReturnTypes.SingleExecutionResult
VAR_INPUT
	(*foreign set to construct substraction*)
	set	: CNM_CollectionInterfaces.ISet;
END_VAR
VAR
	iterator :CNM_CollectionInterfaces.IIterator;
	objectToRemove :CNM_AbstractObject.IObject;
	iteratorState :CNM_ReturnTypes.SingleExecutionState;
END_VAR
instantSubtract := CNM_ReturnTypes.SingleExecutionResult.ABORTED;
RETURN(THIS^.isObjectNull(set) OR_ELSE THIS^.isEqual(set));

instantSubtract := CNM_ReturnTypes.SingleExecutionResult.ERROR;
IF(	set.createNewIterator(iterator => iterator) <> CNM_ReturnTypes.SingleExecutionResult.SUCCESS) THEN
	IF iterator <> 0 THEN
		iterator.destruct();
	END_IF
END_IF

iterator.iterate(FALSE);
instantSubtract := CNM_ReturnTypes.SingleExecutionResult.SUCCESS;
REPEAT 
	iteratorState := iterator.iterate(execute := TRUE, object => objectToRemove); 
	CASE iteratorState OF
	CNM_ReturnTypes.SingleExecutionState.BUSY:
		THIS^.remove(objectToRemove);
	CNM_ReturnTypes.SingleExecutionState.ERROR:
		instantSubtract := CNM_ReturnTypes.SingleExecutionResult.ERROR;
		EXIT;
	END_CASE
UNTIL
	(iteratorState = CNM_ReturnTypes.SingleExecutionState.SUCCESS)
END_REPEAT

iterator.destruct();
END_METHOD

(*

## Short summary

overwrites the content of this set with the intersection of this set and the given set
Set intersection: Common elements between two sets.

**Example:**
Set A = {2, 3, 1, 4}
Set B = {3, 5, 6, 4}

Intersection of A and B: {3, 4}

.. <legal notes>

legal notes
=================
| SPDX-FileCopyrightText: © 2022 ekvip automation GmbH <info@ekvip.de>
| SPDX-License-Identifier: Apache-2.0
| For details check: Apache-2.0_

.. _Apache-2.0: https://www.apache.org/licenses/LICENSE-2.0

.. </legal notes>


**Return:** ``SUCCESS``: if intersect is complete
	``ABORTED``: execute has a falling edge during intersect,
	``BUSY``: Intersect is in Progress
	``ERROR``: the passed collection was not valid or contained invalid Elements or the collection changed during intersect
	``IDLE``: Currently no intersect in progress

*)

METHOD INTERNAL intersect :CNM_ReturnTypes.SingleExecutionState
VAR_INPUT
	(*foreign set to intersect with*)
	set :CNM_CollectionInterfaces.ISet;
	(*If intersect should be processed*)
	execute		:BOOL;
END_VAR
VAR_INST
	cycleManager :CNM_CycleManager.SimpleCycleManager;
	changeIndex :__XWORD;
END_VAR
VAR
	iteratedObject, intersectObject :CNM_AbstractObject.IObject;
	iterateState 				:CNM_ReturnTypes.SingleExecutionState;
	insertOperationsThisCycle	:UDINT := 0;
	objectsRemoved :BOOL := FALSE;
END_VAR
VAR CONSTANT
	INIT :DINT := CNM_ReturnTypes.DefaultSteps.STEP.INIT;
	PROCESSING :DINT := INIT + 1;
	SUCCESS :DINT := CNM_ReturnTypes.DefaultSteps.STEP.SUCCESS;
	ERROR :DINT := CNM_ReturnTypes.DefaultSteps.STEP.ERROR;
END_VAR
REPEAT
	cycleManager(execute := execute);
	CASE cycleManager.step.current OF
	INIT:
		IF THIS^.isObjectValid(THIS^.intersectIterator) THEN 
			THIS^.intersectIterator.destruct();
		END_IF
		IF THIS^.intersectedTree <> 0 THEN
			__DELETE(THIS^.intersectedTree);
		END_IF
		IF (THIS^.isObjectNull(set)) THEN
			cycleManager.proceedWith(ERROR);
			CONTINUE;
		ELSIF (THIS^.isEqual(set)) THEN
			cycleManager.proceedWith(SUCCESS);
			CONTINUE;
		END_IF 
		cycleManager.configuration.sequence.requireSuccessStep := FALSE;
		IF set.size = 0 THEN
			THIS^.clear();
			cycleManager.proceedWith(SUCCESS);
			CONTINUE;
		END_IF
		
		
		IF (set.createNewIterator(iterator => THIS^.intersectIterator) <> CNM_ReturnTypes.SingleExecutionResult.SUCCESS) THEN
			cycleManager.proceedWith(ERROR);
			CONTINUE;	
		END_IF
		THIS^.intersectedTree := __NEW(BalancedBinarySearchTree( nodeComparator := THIS^.nodeComparator));
		IF THIS^.intersectedTree <> 0 THEN
			THIS^.intersectIterator.destruct();
			cycleManager.proceedWith(ERROR);
			CONTINUE;	
		END_IF
		THIS^.intersectIterator.iterate(FALSE);
		cycleManager.proceed();
		
